(* IEC 61131-3 sources: MyTestRepos/BATTERY/PRG, 14 files *)

(* ---- PRG_AI.st ---- *)
PROGRAM PRG_AI
VAR
	F_Trig : ARRAY[1..cnst_num_ai] OF F_TRIG;
	i : INT;	(*Loop variable*)
	ManualFixChannels : BOOL; (*Will reset channels if faulty, i.e. card number is zero*)
	Reset: BOOL;
	Firstrun: BOOL;

	ai_CabinetTemperature_daemon: fb_AiProcess;
	ai_BatteryRoomTemperature_daemon: fb_AiProcess;
	ai_FilterTemperature_daemon: fb_AiProcess;

	ai_CabinetTemperature: str_AiProcess;
	ai_BatteryRoomTemperature: str_AiProcess;
	ai_FilterTemperature: str_AiProcess;

END_VAR

VAR RETAIN
	ai_CabinetTemperature_setup: str_AiSetup;
	ai_BatteryRoomTemperature_setup: str_AiSetup;
	ai_FilterTemperature_setup: str_AiSetup;
END_VAR

Reset := PRG_Functions.Reset;

(*Setup the HMI variables so that they are equal to actual used variables*)
IF (NOT Firstrun) THEN
	hmi_AiSetup[1] := ai_CabinetTemperature_setup;
	hmi_AiSetup[2] := ai_BatteryRoomTemperature_setup;
	hmi_AiSetup[3] := ai_FilterTemperature_setup;
	Firstrun := TRUE;
END_IF

(*Analog Input Signals*)
	ai_CabinetTemperature_daemon (setup:=ai_CabinetTemperature_setup,reset:=Reset,outPV=>ai_CabinetTemperature);
	ai_BatteryRoomTemperature_daemon (setup:=ai_BatteryRoomTemperature_setup,reset:=Reset,outPV=>ai_BatteryRoomTemperature);
	ai_FilterTemperature_daemon (setup:=ai_FilterTemperature_setup,reset:=Reset,outPV=>ai_FilterTemperature);

(*HMI Assign*)
	hmi_AiPV[1]:=ai_CabinetTemperature_daemon.outPV;
	hmi_AiPV[2]:=ai_BatteryRoomTemperature_daemon.outPV;
	hmi_AiPV[3]:=ai_FilterTemperature_daemon.outPV;

IF (ManualFixChannels) THEN  (*If manually forced: re-configure the channels*)
	FOR i:=0 TO cnst_num_ai BY 1 DO				(*Check if channel info is empty and restore if so.*)
		IF (PRG_HMI.setup_AioCard1_Number <> 0) THEN
			hmi_RestoreDefault_ai[i] := TRUE;
		END_IF
	END_FOR;
	ManualFixChannels := FALSE;
END_IF

END_PROGRAM

ACTIONS

ACTION Settings
(*
THIS SECTION CONTAINS HARD-CODED CHANNEL SETTINGS FOR EACH OF THE ANALOG INPUTS.

The settings are stored in retain memory, but whenever permanent changes are made, they should be hard coded into the appropriate channel below.
Each channel has settings for:

- Channel name (used for presentation in HMI)
- Channel- and card number (used to retrieve channel value via MIO lib)
- Channel type (4-20mA, PT100 etc)
- Channel forcing (force value and a bool flag to enable/disable forcing)
- Channel error flags, along with enable/disable flag + time delays
- Channel level flags, along with enable/disable flag + time delays

All setup values in retain memory can be forced to default (hard coded) values by setting RestoreAllToDefault,
or individually by setting hmi_RestoreDefault_ai[]. The latter is primary used from HMI.
*)
(***************ai_CabinetTemperature***************)
IF (RestoreAllToDefault OR ai_CabinetTemperature_setup.RestoreDefault  OR hmi_RestoreDefault_ai[1]) THEN
	ai_CabinetTemperature_setup.Name:='ai_CabinetTemperature';
	ai_CabinetTemperature_setup.CardNb:=PRG_HMI.setup_AioCard1_Number;
	ai_CabinetTemperature_setup.ChannelMode:=16#D3;
	ai_CabinetTemperature_setup.ChannelNb:=1;
 	ai_CabinetTemperature_setup.Enable.Forcing:=0;
 	ai_CabinetTemperature_setup.Enable.LLL:=0;
 	ai_CabinetTemperature_setup.Enable.LL:=0;
 	ai_CabinetTemperature_setup.Enable.L:=0;
 	ai_CabinetTemperature_setup.Enable.H:=0;
 	ai_CabinetTemperature_setup.Enable.HH:=0;
 	ai_CabinetTemperature_setup.Enable.HHH:=0;
 	ai_CabinetTemperature_setup.Enable.WireBreak:=1;
 	ai_CabinetTemperature_setup.Enable.Freeze:=1;
 	ai_CabinetTemperature_setup.Enable.High:=1;
 	ai_CabinetTemperature_setup.Enable.OOR:=1;
 	ai_CabinetTemperature_setup.Delay.LLL:=T#1s;
 	ai_CabinetTemperature_setup.Delay.LL:=T#1s;
 	ai_CabinetTemperature_setup.Delay.L:=T#1s;
 	ai_CabinetTemperature_setup.Delay.H:=T#1s;
 	ai_CabinetTemperature_setup.Delay.HH:=T#1s;
 	ai_CabinetTemperature_setup.Delay.HHH:=T#1s;
 	ai_CabinetTemperature_setup.Delay.WireBreak:=T#1s;
 	ai_CabinetTemperature_setup.Delay.High:=T#1s;
 	ai_CabinetTemperature_setup.Delay.OOR:=T#1s;
 	ai_CabinetTemperature_setup.Levels.LLL:=0;
 	ai_CabinetTemperature_setup.Levels.LL:=0;
 	ai_CabinetTemperature_setup.Levels.L:=0;
 	ai_CabinetTemperature_setup.Levels.H:=0;
 	ai_CabinetTemperature_setup.Levels.HH:=0;
 	ai_CabinetTemperature_setup.Levels.HHH:=0;
 	ai_CabinetTemperature_setup.Levels.Scale4mA:=0;
 	ai_CabinetTemperature_setup.Levels.Scale20mA:=100;
 	ai_CabinetTemperature_setup.Levels.ForceValue:=0;
END_IF
IF (hmi_RestoreDefault_ai[1] OR RestoreAllToDefault OR ai_CabinetTemperature_setup.RestoreDefault) THEN (*Copy values into HMI variable and reset*)
	hmi_AiSetup[1]:=ai_CabinetTemperature_setup; (*Copy setup values from retain into hmi variable*)
	hmi_RestoreDefault_ai[1]:=FALSE; (*Make sure that the restore variable is turned off after one restore command*)
	ai_CabinetTemperature_setup.RestoreDefault:=FALSE; (*Make sure that the restore variable is turned off after one restore command*)
END_IF
IF (hmi_AiWriteSetup[1]) THEN
	ai_CabinetTemperature_setup:=hmi_AiSetup[1]; (*Paste hmi changes back into setup variable*)
	hmi_AiWriteSetup[1]:=FALSE; (*Make sure that the write variable is turned off after one write command*)
END_IF
F_Trig[1](CLK:=hmi_AiPV[1].IsForced); (*Reset HMI forcing dialog when timer runs out*)
IF (F_Trig[1].Q) THEN hmi_AiSetup[1].Enable.Forcing:=FALSE;ai_CabinetTemperature_setup.Enable.Forcing:=FALSE; END_IF
(**************************************************)

(***************ai_BatteryRoomTemperature***************)
IF (RestoreAllToDefault OR ai_BatteryRoomTemperature_setup.RestoreDefault  OR hmi_RestoreDefault_ai[2]) THEN
	ai_BatteryRoomTemperature_setup.Name:='ai_BatteryRoomTemperature';
	ai_BatteryRoomTemperature_setup.CardNb:=PRG_HMI.setup_AioCard1_Number;
	ai_BatteryRoomTemperature_setup.ChannelMode:=16#D3;
	ai_BatteryRoomTemperature_setup.ChannelNb:=2;
 	ai_BatteryRoomTemperature_setup.Enable.Forcing:=0;
 	ai_BatteryRoomTemperature_setup.Enable.LLL:=0;
 	ai_BatteryRoomTemperature_setup.Enable.LL:=0;
 	ai_BatteryRoomTemperature_setup.Enable.L:=0;
 	ai_BatteryRoomTemperature_setup.Enable.H:=0;
 	ai_BatteryRoomTemperature_setup.Enable.HH:=0;
 	ai_BatteryRoomTemperature_setup.Enable.HHH:=0;
 	ai_BatteryRoomTemperature_setup.Enable.WireBreak:=1;
 	ai_BatteryRoomTemperature_setup.Enable.Freeze:=1;
 	ai_BatteryRoomTemperature_setup.Enable.High:=1;
 	ai_BatteryRoomTemperature_setup.Enable.OOR:=1;
 	ai_BatteryRoomTemperature_setup.Delay.LLL:=T#1s;
 	ai_BatteryRoomTemperature_setup.Delay.LL:=T#1s;
 	ai_BatteryRoomTemperature_setup.Delay.L:=T#1s;
 	ai_BatteryRoomTemperature_setup.Delay.H:=T#1s;
 	ai_BatteryRoomTemperature_setup.Delay.HH:=T#1s;
 	ai_BatteryRoomTemperature_setup.Delay.HHH:=T#1s;
 	ai_BatteryRoomTemperature_setup.Delay.WireBreak:=T#1s;
 	ai_BatteryRoomTemperature_setup.Delay.High:=T#1s;
 	ai_BatteryRoomTemperature_setup.Delay.OOR:=T#1s;
 	ai_BatteryRoomTemperature_setup.Levels.LLL:=0;
 	ai_BatteryRoomTemperature_setup.Levels.LL:=0;
 	ai_BatteryRoomTemperature_setup.Levels.L:=0;
 	ai_BatteryRoomTemperature_setup.Levels.H:=0;
 	ai_BatteryRoomTemperature_setup.Levels.HH:=0;
 	ai_BatteryRoomTemperature_setup.Levels.HHH:=0;
 	ai_BatteryRoomTemperature_setup.Levels.Scale4mA:=-20;
 	ai_BatteryRoomTemperature_setup.Levels.Scale20mA:=80;
 	ai_BatteryRoomTemperature_setup.Levels.ForceValue:=0;
END_IF
IF (hmi_RestoreDefault_ai[2] OR RestoreAllToDefault OR ai_BatteryRoomTemperature_setup.RestoreDefault) THEN (*Copy values into HMI variable and reset*)
	hmi_AiSetup[2]:=ai_BatteryRoomTemperature_setup; (*Copy setup values from retain into hmi variable*)
	hmi_RestoreDefault_ai[2]:=FALSE; (*Make sure that the restore variable is turned off after one restore command*)
	ai_BatteryRoomTemperature_setup.RestoreDefault:=FALSE; (*Make sure that the restore variable is turned off after one restore command*)
END_IF
IF (hmi_AiWriteSetup[2]) THEN
	ai_BatteryRoomTemperature_setup:=hmi_AiSetup[2]; (*Paste hmi changes back into setup variable*)
	hmi_AiWriteSetup[2]:=FALSE; (*Make sure that the write variable is turned off after one write command*)
END_IF
F_Trig[2](CLK:=hmi_AiPV[2].IsForced); (*Reset HMI forcing dialog when timer runs out*)
IF (F_Trig[2].Q) THEN hmi_AiSetup[2].Enable.Forcing:=FALSE;ai_BatteryRoomTemperature_setup.Enable.Forcing:=FALSE; END_IF
(**************************************************)

(***************ai_FilterTemperature***************)
IF (RestoreAllToDefault OR ai_FilterTemperature_setup.RestoreDefault  OR hmi_RestoreDefault_ai[3]) THEN
	ai_FilterTemperature_setup.Name:='ai_FilterTemperature';
	ai_FilterTemperature_setup.CardNb:=PRG_HMI.setup_AioCard1_Number;
	ai_FilterTemperature_setup.ChannelMode:=16#D1;
	ai_FilterTemperature_setup.ChannelNb:=4;
 	ai_FilterTemperature_setup.Enable.Forcing:=0;
 	ai_FilterTemperature_setup.Enable.LLL:=0;
 	ai_FilterTemperature_setup.Enable.LL:=0;
 	ai_FilterTemperature_setup.Enable.L:=0;
 	ai_FilterTemperature_setup.Enable.H:=0;
 	ai_FilterTemperature_setup.Enable.HH:=0;
 	ai_FilterTemperature_setup.Enable.HHH:=0;
 	ai_FilterTemperature_setup.Enable.WireBreak:=1;
 	ai_FilterTemperature_setup.Enable.Freeze:=1;
 	ai_FilterTemperature_setup.Enable.High:=1;
 	ai_FilterTemperature_setup.Enable.OOR:=1;
 	ai_FilterTemperature_setup.Delay.LLL:=T#1s;
 	ai_FilterTemperature_setup.Delay.LL:=T#1s;
 	ai_FilterTemperature_setup.Delay.L:=T#1s;
 	ai_FilterTemperature_setup.Delay.H:=T#1s;
 	ai_FilterTemperature_setup.Delay.HH:=T#1s;
 	ai_FilterTemperature_setup.Delay.HHH:=T#1s;
 	ai_FilterTemperature_setup.Delay.WireBreak:=T#1s;
 	ai_FilterTemperature_setup.Delay.High:=T#1s;
 	ai_FilterTemperature_setup.Delay.OOR:=T#1s;
 	ai_FilterTemperature_setup.Levels.LLL:=0;
 	ai_FilterTemperature_setup.Levels.LL:=0;
 	ai_FilterTemperature_setup.Levels.L:=0;
 	ai_FilterTemperature_setup.Levels.H:=0;
 	ai_FilterTemperature_setup.Levels.HH:=0;
 	ai_FilterTemperature_setup.Levels.HHH:=0;
 	ai_FilterTemperature_setup.Levels.Scale4mA:=0;
 	ai_FilterTemperature_setup.Levels.Scale20mA:=100;
 	ai_FilterTemperature_setup.Levels.ForceValue:=0;
END_IF
IF (hmi_RestoreDefault_ai[3] OR RestoreAllToDefault OR ai_FilterTemperature_setup.RestoreDefault) THEN (*Copy values into HMI variable and reset*)
	hmi_AiSetup[3]:=ai_FilterTemperature_setup; (*Copy setup values from retain into hmi variable*)
	hmi_RestoreDefault_ai[3]:=FALSE; (*Make sure that the restore variable is turned off after one restore command*)
	ai_FilterTemperature_setup.RestoreDefault:=FALSE; (*Make sure that the restore variable is turned off after one restore command*)
END_IF
IF (hmi_AiWriteSetup[3]) THEN
	ai_FilterTemperature_setup:=hmi_AiSetup[3]; (*Paste hmi changes back into setup variable*)
	hmi_AiWriteSetup[3]:=FALSE; (*Make sure that the write variable is turned off after one write command*)
END_IF
F_Trig[3](CLK:=hmi_AiPV[3].IsForced); (*Reset HMI forcing dialog when timer runs out*)
IF (F_Trig[3].Q) THEN hmi_AiSetup[3].Enable.Forcing:=FALSE;ai_FilterTemperature_setup.Enable.Forcing:=FALSE; END_IF
(**************************************************)

END_ACTION

END_ACTIONS

(* ---- PRG_Alarms.st ---- *)
PROGRAM PRG_Alarms
VAR
	pack: 					INT := 0;
	BMS_Alarm_Word: 		INT := 8; (*Must be first available word number after the ordinary alarms*)

	(*Two dimensional array for Set/Reset blocks. First index refers to word number (e.g. Alarmword[1]), second index refers to bit number*)
	AlarmSR: 				ARRAY[1..32,0..15] OF SR;
	Repeat_Alarm: 			fb_RepeatAlarm;
	Repeat_AlarmAppWarning:	fb_RepeatAlarm;
	E0AlarmWord:			fb_BitToWord;

	Reset : 				BOOL;
	CommonWarning: 			BOOL;
	CommonPLCWarning:		BOOL;
	CommonAppWarning:		BOOL;
	CommonIoWarning:		BOOL;
	CommonLevelWarning:		BOOL;
	CommonSignalWarning:	BOOL;
	CommonE0Warning:		BOOL;
END_VAR

Reset := PRG_Functions.Reset;

(*Gorup alarms with blinking on new alarms within their group*)
CommonWarning :=  		Repeat_Alarm.Alarm_common;
CommonPLCWarning := 	Repeat_Alarm.Alarm_Repeat1;
CommonSignalWarning:= 	Repeat_Alarm.Alarm_Repeat2;
CommonIoWarning	 := 	Repeat_Alarm.Alarm_Repeat3;
CommonLevelWarning := 	Repeat_Alarm.Alarm_Repeat4;
CommonAppWarning := 	Repeat_AlarmAppWarning.Alarm_common;
CommonE0Warning := 		Repeat_Alarm.Alarm_Repeat20;

(*Single alarms used for E0 *)
E0AlarmWord(
	EN := TRUE,
	Bit0 := PRG_DI.di_WaterLeakageDetected.PV,
	Bit1 := PRG_BatteryProtection.batteryPreWarning,
	Bit2 := PRG_BatteryProtection.Warning_CellTemp_L,
	Bit3 := PRG_BatteryProtection.Warning_CellVolt_L_Offline,
	Bit4 := PRG_BatteryProtection.Warning_CellVolt_LL_Offline,
	Bit5 := PRG_BatteryProtection.Warning_SoC_L_Offline,
	Bit6 := FALSE,
	Bit7 := FALSE,
	Bit8 := FALSE,
	Bit9 := FALSE,
	Bit10 := FALSE,
	Bit11 := FALSE,
	Bit12 := FALSE,
	Bit13 := FALSE,
	Bit14 := FALSE,
	Bit15 := FALSE,
	OUT =>
);

(*General PLC warnings*)
AlarmSR[1,0] (SET1:=(PRG_HW.HwAlarmCPU.AlarmCpuLoad) ,  Q1=>AlarmWord[1].0, RESET:=PRG_Functions.Reset);(*High Load on CPU*)
AlarmSR[1,1] (SET1:=(PRG_HW.HwAlarmCPU.AlarmCpuTemp) ,  Q1=>AlarmWord[1].1, RESET:=PRG_Functions.Reset);(*High Temperature on CPU*)
AlarmSR[1,2] (SET1:=(PRG_HW.HwAlarmCPU.AlarmFreeMem) ,  Q1=>AlarmWord[1].2, RESET:=PRG_Functions.Reset);(*Low Free Memory on PLC CPU*)
AlarmSR[1,3] (SET1:=(PRG_HW.Em0In.Alarm) ,  Q1=>AlarmWord[1].3, RESET:=PRG_Functions.Reset);(*High Load on EM213 Network Card*)
AlarmSR[1,4] (SET1:=(PRG_HW.Eth0In.Alarm) ,  Q1=>AlarmWord[1].4, RESET:=PRG_Functions.Reset);(*High Load on Ethernet Port ETH1*)
AlarmSR[1,5] (SET1:=(PRG_HW.Eth1In.Alarm) ,  Q1=>AlarmWord[1].5, RESET:=PRG_Functions.Reset);(*High Load on Ethernet Port ETH2*)

(*Signal warnings, OOR and wirebreak etc*)
AlarmSR[2,0] (SET1:=(PRG_AI.ai_BatteryRoomTemperature.Alarm.common) ,  Q1=>AlarmWord[2].0, RESET:=PRG_Functions.Reset);(*Battery Room Temperature - 4mA loop fail*)
AlarmSR[2,1] (SET1:=(PRG_AI.ai_CabinetTemperature.Alarm.common) ,  Q1=>AlarmWord[2].1, RESET:=PRG_Functions.Reset);(*Cabinet Temperature - Loop Failure*)
AlarmSR[2,2] (SET1:=(PRG_AI.ai_FilterTemperature.Alarm.common) ,  Q1=>AlarmWord[2].2, RESET:=PRG_Functions.Reset);(*LC Filter Temperature - Loop Failure*)
AlarmSR[2,3] (SET1:=(PRG_AO.ao_BatteryCurrentInstr.Alarm.common) ,  Q1=>AlarmWord[2].3, RESET:=PRG_Functions.Reset);(*Current Instrument 4-20mA Loop Failure*)
AlarmSR[2,4] (SET1:=(PRG_AO.ao_BatteryPowerInstr.Alarm.common) ,  Q1=>AlarmWord[2].4, RESET:=PRG_Functions.Reset);(*Power Instrument 4-20mA Loop Failure*)
AlarmSR[2,5] (SET1:=(PRG_AO.ao_BatteryVoltageInstr.Alarm.common) ,  Q1=>AlarmWord[2].5, RESET:=PRG_Functions.Reset);(*Voltage Instrument 4-20mA Loop Failure*)
AlarmSR[2,6] (SET1:=(PRG_AO.ao_BatterySocInstr.Alarm.common) ,  Q1=>AlarmWord[2].6, RESET:=PRG_Functions.Reset);(*SoC Instrument 4-20mA Loop Failure*)
AlarmSR[2,7] (SET1:=(PRG_AO.ao_BatteryChrgDischrgInstr.Alarm.common) ,  Q1=>AlarmWord[2].7, RESET:=PRG_Functions.Reset);(*Charge/Discharge Instrument 4-20mA Loop Failure*)

(*IO warnings, alarm contacts, module error etc*)
AlarmSR[3,0] (SET1:=(PRG_HW.AioCardError1) ,  Q1=>AlarmWord[3].0, RESET:=PRG_Functions.Reset);(*Common Alarm from PLC I/O Analog IO Card*)
AlarmSR[3,1] (SET1:=(PRG_HW.DioCardError1) ,  Q1=>AlarmWord[3].1, RESET:=PRG_Functions.Reset);(*Common Alarm from PLC I/O Digital IO Card*)
AlarmSR[3,2] (SET1:=(PRG_Functions.Breaker.Alarm_delayed) ,  Q1=>AlarmWord[3].2, RESET:=PRG_Functions.Reset);(*Voting Alarm DC Breaker Position*)
AlarmSR[3,3] (SET1:=(PRG_DI.di_EmergencyStopLoopFault.PV) ,  Q1=>AlarmWord[3].3, RESET:=PRG_Functions.Reset);(*Emergency Stop Loop Alarm*)
AlarmSR[3,4] (SET1:=(PRG_Operation.ControlPlace.alarmDeviation) ,  Q1=>AlarmWord[3].4, RESET:=PRG_Functions.Reset);(*Voting Alarm Local/Remote Switch*)
AlarmSR[3,5] (SET1:=(NOT PRG_DI.di_EthernetSwitchAlarm.PV AND PRG_HMI.enEthernetSwitchAlarm) ,  Q1=>AlarmWord[3].5, RESET:=PRG_Functions.Reset);(*External Ethernet Switch Alarm*)

(*Level warning, high or low etc*)
AlarmSR[4,0] (SET1:=(PRG_AI.ai_BatteryRoomTemperature.Alarm.HH) ,  Q1=>AlarmWord[4].0, RESET:=PRG_Functions.Reset);(*Battery Room High Temperature*)
AlarmSR[4,1] (SET1:=(PRG_AI.ai_BatteryRoomTemperature.Alarm.LL) ,  Q1=>AlarmWord[4].1, RESET:=PRG_Functions.Reset);(*Battery Room Low Temperature*)
AlarmSR[4,2] (SET1:=(PRG_AI.ai_BatteryRoomTemperature.Alarm.HHH) ,  Q1=>AlarmWord[4].2, RESET:=PRG_Functions.Reset);(*Battery Room HighHigh Temperature*)
AlarmSR[4,3] (SET1:=(PRG_AI.ai_BatteryRoomTemperature.Alarm.LLL) ,  Q1=>AlarmWord[4].3, RESET:=PRG_Functions.Reset);(*Battery Room LowLow Temperature*)
AlarmSR[4,4] (SET1:=(PRG_AI.ai_CabinetTemperature.Alarm.HH) ,  Q1=>AlarmWord[4].4, RESET:=PRG_Functions.Reset);(*Cabinet High Temperature*)
AlarmSR[4,5] (SET1:=(PRG_AI.ai_CabinetTemperature.Alarm.LL) ,  Q1=>AlarmWord[4].5, RESET:=PRG_Functions.Reset);(*Cabinet Low Temperature*)
AlarmSR[4,6] (SET1:=(PRG_AI.ai_FilterTemperature.Alarm.HH) ,  Q1=>AlarmWord[4].6, RESET:=PRG_Functions.Reset);(*LC Filter High Temperature*)
AlarmSR[4,7] (SET1:=(PRG_AI.ai_FilterTemperature.Alarm.LL) ,  Q1=>AlarmWord[4].7, RESET:=PRG_Functions.Reset);(*LC Filter Low Temperature*)
AlarmSR[4,8] (SET1:=(PRG_Drive.UnitOverTempAlarm) ,  Q1=>AlarmWord[4].8, RESET:=PRG_Functions.Reset);(*Vacon Unit High Temperature*)

(*Application specific warnings*)
AlarmSR[5,0] (SET1:=(PRG_Drive.Status.Warning) ,  Q1=>AlarmWord[5].0, RESET:=PRG_Functions.Reset);(*Common Alarm from DC/DC Converter*)
AlarmSR[5,1] (SET1:=(PRG_BatteryProtection.batteryCommonWarning) ,  Q1=>AlarmWord[5].1, RESET:=PRG_Functions.Reset);(*Common Alarm from Battery Management System*)
AlarmSR[5,2] (SET1:=(PRG_StateMain.StartingTimeout) ,  Q1=>AlarmWord[5].2, RESET:=PRG_Functions.Reset);(*Start Sequence Timeout*)
AlarmSR[5,3] (SET1:=(PRG_StateMain.StoppingTimeout) ,  Q1=>AlarmWord[5].3, RESET:=PRG_Functions.Reset);(*Stop Sequence Timeout - Failsafe Trip*)
AlarmSR[5,4] (SET1:=(PRG_DI.di_WaterLeakageDetected.PV) ,  Q1=>AlarmWord[5].4, RESET:=PRG_Functions.Reset);(*Water Leakage in DC/DC Section*)
AlarmSR[5,5] (SET1:=(PRG_Battery.StopChargeTOF.Q) ,  Q1=>AlarmWord[5].5, RESET:=PRG_Functions.Reset);(*Battery Charge Limit in Effect*)
AlarmSR[5,6] (SET1:=(PRG_Battery.StopDischargeTOF.Q) ,  Q1=>AlarmWord[5].6, RESET:=PRG_Functions.Reset);(*Battery Discharge Limit in Effect*)
AlarmSR[5,7] (SET1:=(NOT PRG_Functions.Breaker.DI_Verif_delay OR NOT PRG_DI.di_DcBreakerEarlyBreak.PV) ,  Q1=>AlarmWord[5].7, RESET:=PRG_Functions.Reset);(*DC Breaker Open - Start Inhibited*)
AlarmSR[5,8] (SET1:=(PRG_Operation.ControlPlace.ctrlLocation = e_Local) ,  Q1=>AlarmWord[5].8, RESET:=PRG_Functions.Reset);(*In Local Control*)
AlarmSR[5,9] (SET1:=(PRG_IAS.IasCommunication.Alarm) ,  Q1=>AlarmWord[5].9, RESET:=PRG_Functions.Reset);(*IAS Communication Alarm*)
AlarmSR[5,10] (SET1:=(PRG_BatteryComm.NoPrechargePackComm) ,  Q1=>AlarmWord[5].10, RESET:=PRG_Functions.Reset);(*Comm. Failure Battery Precharge System*)
AlarmSR[5,11] (SET1:=((PRG_StateMain.RunningTON.Q) AND NOT PRG_Battery.BatteryAllConnected) ,  Q1=>AlarmWord[5].11, RESET:=PRG_Functions.Reset);(*All Batteries are not Connected*)
AlarmSR[5,12] (SET1:=(PRG_StateMain.BatteryConnectionTimeout) ,  Q1=>AlarmWord[5].12, RESET:=PRG_Functions.Reset);(*Battery Connection Timeout during Starting*)
AlarmSR[5,13] (SET1:=(PRG_StateMain.BatteryDisconnectionTimeout) ,  Q1=>AlarmWord[5].13, RESET:=PRG_Functions.Reset);(*Battery Disconnection Timeout during Stopping*)

(*Battery Specific PLC Alarms*)
AlarmSR[6,0] (SET1:=(PRG_BatteryProtection.batteryPreWarning) ,  Q1=>AlarmWord[6].0, RESET:=PRG_Functions.Reset);(*Prewarning from Battery Management System*)
AlarmSR[6,1] (SET1:=(PRG_BatteryProtection.Warning_SoC_L) ,  Q1=>AlarmWord[6].1, RESET:=PRG_Functions.Reset);(*State of Charge Low Alarm - Start Charging*)
AlarmSR[6,2] (SET1:=(PRG_BatteryProtection.Warning_SoC_H) ,  Q1=>AlarmWord[6].2, RESET:=PRG_Functions.Reset);(*State of Charge High Alarm*)
AlarmSR[6,3] (SET1:=(PRG_BatteryProtection.Warning_Volt_H) ,  Q1=>AlarmWord[6].3, RESET:=PRG_Functions.Reset);(*High Battery Voltage Alarm*)
AlarmSR[6,4] (SET1:=(PRG_BatteryProtection.Warning_Volt_L) ,  Q1=>AlarmWord[6].4, RESET:=PRG_Functions.Reset);(*Low Battery Voltage Alarm*)
AlarmSR[6,5] (SET1:=(PRG_BatteryProtection.Warning_CellVolt_L) ,  Q1=>AlarmWord[6].5, RESET:=PRG_Functions.Reset);(*Low Cell Voltage Alarm*)
AlarmSR[6,6] (SET1:=(PRG_BatteryProtection.Warning_CellVolt_H) ,  Q1=>AlarmWord[6].6, RESET:=PRG_Functions.Reset);(*High Cell Voltage Alarm*)
AlarmSR[6,7] (SET1:=(PRG_BatteryProtection.Warning_CellTemp_L) ,  Q1=>AlarmWord[6].7, RESET:=PRG_Functions.Reset);(*Low Cell Temperature Alarm*)
AlarmSR[6,8] (SET1:=(PRG_BatteryProtection.Warning_CellTemp_H) ,  Q1=>AlarmWord[6].8, RESET:=PRG_Functions.Reset);(*High Cell Temperature Alarm*)
AlarmSR[6,9] (SET1:=(PRG_BatteryProtection.Warning_SoC_L_Offline) ,  Q1=>AlarmWord[6].9, RESET:=PRG_Functions.Reset);(*Offline Low SoC: Connect and Charge Now*)
AlarmSR[6,10] (SET1:=(PRG_BatteryProtection.Warning_CellVolt_L_Offline) ,  Q1=>AlarmWord[6].10, RESET:=PRG_Functions.Reset);(*Offline Low Cell Voltage: Connect and Charge Now*)
AlarmSR[6,11] (SET1:=(PRG_BatteryProtection.Warning_CellVolt_LL_Offline) ,  Q1=>AlarmWord[6].11, RESET:=PRG_Functions.Reset);(*Offline Low Cell Voltage: Critical Level - Charge Now*)
AlarmSR[6,12] (SET1:=(PRG_HMI.SoHVerifModeActive) ,  Q1=>AlarmWord[6].12, RESET:=PRG_Functions.Reset);(*SoH Verification Mode Active: SoC Limits Extended*)

(*Auto generated alarms from Corvus BMS*)

BMS_Alarm_Word:= 8; (*Next available alarmword*)
FOR pack := 1 TO DINT_TO_INT(PRG_HMI.setup_Battery_total_nr_of_packs) BY 1 DO
	AlarmSR[BMS_Alarm_Word,0] (SET1:=(PRG_BatteryComm.CorvusRead[pack].FW.Input_PowerLoss_Warning) ,  Q1=>AlarmWord[BMS_Alarm_Word].0, RESET:=Reset);(*BMS Pack  Input Power Loss Warning*)
	AlarmSR[BMS_Alarm_Word,1] (SET1:=(PRG_BatteryComm.CorvusRead[pack].FW.Module_Communication_Warning) ,  Q1=>AlarmWord[BMS_Alarm_Word].1, RESET:=Reset);(*BMS Pack  Module Communication Warning*)
	AlarmSR[BMS_Alarm_Word,2] (SET1:=(PRG_BatteryComm.CorvusRead[pack].FW.OverCurrent_Warning) ,  Q1=>AlarmWord[BMS_Alarm_Word].2, RESET:=Reset);(*BMS Pack  Over Current Warning*)
	AlarmSR[BMS_Alarm_Word,3] (SET1:=(PRG_BatteryComm.CorvusRead[pack].FW.PDM_overTemperature_Warning) ,  Q1=>AlarmWord[BMS_Alarm_Word].3, RESET:=Reset);(*BMS Pack  PDM Over Temperature Warning*)
	AlarmSR[BMS_Alarm_Word,4] (SET1:=(PRG_BatteryComm.CorvusRead[pack].FW.SE_overTemperature_Warning) ,  Q1=>AlarmWord[BMS_Alarm_Word].4, RESET:=Reset);(*BMS Pack  Cell Over Temperature Warning*)
	AlarmSR[BMS_Alarm_Word,5] (SET1:=(PRG_BatteryComm.CorvusRead[pack].FW.SE_overVoltage_Warning) ,  Q1=>AlarmWord[BMS_Alarm_Word].5, RESET:=Reset);(*BMS Pack  Cell Over Voltage Warning*)
	AlarmSR[BMS_Alarm_Word,6] (SET1:=(PRG_BatteryComm.CorvusRead[pack].FW.SE_underVoltage_Warning) ,  Q1=>AlarmWord[BMS_Alarm_Word].6, RESET:=Reset);(*BMS Pack  Cell Under Voltage Warning*)
	AlarmSR[BMS_Alarm_Word,7] (SET1:=(PRG_BatteryComm.CorvusRead[pack].ModbusFault AND NOT PRG_BatteryComm.CorvusBMS_Total_Comm_Fault) ,  Q1=>AlarmWord[BMS_Alarm_Word].7, RESET:=Reset);(*BMS Pack Communication Alarm*)
	BMS_Alarm_Word :=  BMS_Alarm_Word+1;
END_FOR

(*Blinks the alarm output*)

Repeat_AlarmAppWarning(
	AlarmWord5:= INT_TO_WORD(AlarmWord[5]),
	AlarmWord6:= INT_TO_WORD(AlarmWord[6]),
);

Repeat_Alarm(
	AlarmWord1:= INT_TO_WORD(AlarmWord[1]),
	AlarmWord2:= INT_TO_WORD(AlarmWord[2]),
	AlarmWord3:= INT_TO_WORD(AlarmWord[3]),
	AlarmWord4:= INT_TO_WORD(AlarmWord[4]),
	AlarmWord5:= INT_TO_WORD(AlarmWord[5]),
	AlarmWord6:= INT_TO_WORD(AlarmWord[6]),
	AlarmWord7:= INT_TO_WORD(AlarmWord[7]),
	AlarmWord8:= INT_TO_WORD(AlarmWord[8]),
	AlarmWord9:= INT_TO_WORD(AlarmWord[9]),
	AlarmWord10:= INT_TO_WORD(AlarmWord[10]),
	AlarmWord11:= INT_TO_WORD(AlarmWord[11]),
	AlarmWord12:= INT_TO_WORD(AlarmWord[12]),
	AlarmWord13:= INT_TO_WORD(AlarmWord[13]),
	AlarmWord14:= INT_TO_WORD(AlarmWord[14]),
	AlarmWord15:= INT_TO_WORD(AlarmWord[15]),
	AlarmWord16:= INT_TO_WORD(AlarmWord[16]),
	AlarmWord17:= INT_TO_WORD(AlarmWord[17]),
	AlarmWord18:= INT_TO_WORD(AlarmWord[18]),
	AlarmWord19:= INT_TO_WORD(AlarmWord[19]),
	AlarmWord20:= DINT_TO_WORD(E0AlarmWord.OUT),
	Alarm_common => ,
	Alarm_count => ,
	Alarm_Repeat1 => ,
	Alarm_Repeat2 => ,
	Alarm_Repeat3 => ,
	Alarm_Repeat4 => ,
	Alarm_Repeat5 => ,
	Alarm_Repeat6 => ,
	Alarm_Repeat7 => ,
	Alarm_Repeat8 => ,
	Alarm_Repeat9 => ,
	Alarm_Repeat10 => ,
	Alarm_Repeat11 => ,
	Alarm_Repeat12 => ,
	Alarm_Repeat13 => ,
	Alarm_Repeat14 => ,
	Alarm_Repeat15 => ,
	Alarm_Repeat16 => ,
	Alarm_Repeat17 => ,
	Alarm_Repeat18 => ,
	Alarm_Repeat19 => ,
	Alarm_Repeat20 =>
);

END_PROGRAM

ACTIONS
ACTION hmi_Alarms
hmi_AlarmWord[1].0 := AlarmSR[1,0].Q1;
hmi_AlarmWord[1].1 := AlarmSR[1,1].Q1;
hmi_AlarmWord[1].2 := AlarmSR[1,2].Q1;
hmi_AlarmWord[1].3 := AlarmSR[1,3].Q1;
hmi_AlarmWord[1].4 := AlarmSR[1,4].Q1;
hmi_AlarmWord[1].5 := AlarmSR[1,5].Q1;
hmi_AlarmWord[1].6 := AlarmSR[1,6].Q1;
hmi_AlarmWord[1].7 := AlarmSR[1,7].Q1;
hmi_AlarmWord[1].8 := AlarmSR[1,8].Q1;
hmi_AlarmWord[1].9 := AlarmSR[1,9].Q1;
hmi_AlarmWord[1].10 := AlarmSR[1,10].Q1;
hmi_AlarmWord[1].11 := AlarmSR[1,11].Q1;
hmi_AlarmWord[1].12 := AlarmSR[1,12].Q1;
hmi_AlarmWord[1].13 := AlarmSR[1,13].Q1;
hmi_AlarmWord[1].14 := AlarmSR[1,14].Q1;
hmi_AlarmWord[1].15 := AlarmSR[1,15].Q1;
hmi_AlarmWord[2].0 := AlarmSR[2,0].Q1;
hmi_AlarmWord[2].1 := AlarmSR[2,1].Q1;
hmi_AlarmWord[2].2 := AlarmSR[2,2].Q1;
hmi_AlarmWord[2].3 := AlarmSR[2,3].Q1;
hmi_AlarmWord[2].4 := AlarmSR[2,4].Q1;
hmi_AlarmWord[2].5 := AlarmSR[2,5].Q1;
hmi_AlarmWord[2].6 := AlarmSR[2,6].Q1;
hmi_AlarmWord[2].7 := AlarmSR[2,7].Q1;
hmi_AlarmWord[2].8 := AlarmSR[2,8].Q1;
hmi_AlarmWord[2].9 := AlarmSR[2,9].Q1;
hmi_AlarmWord[2].10 := AlarmSR[2,10].Q1;
hmi_AlarmWord[2].11 := AlarmSR[2,11].Q1;
hmi_AlarmWord[2].12 := AlarmSR[2,12].Q1;
hmi_AlarmWord[2].13 := AlarmSR[2,13].Q1;
hmi_AlarmWord[2].14 := AlarmSR[2,14].Q1;
hmi_AlarmWord[2].15 := AlarmSR[2,15].Q1;
hmi_AlarmWord[3].0 := AlarmSR[3,0].Q1;
hmi_AlarmWord[3].1 := AlarmSR[3,1].Q1;
hmi_AlarmWord[3].2 := AlarmSR[3,2].Q1;
hmi_AlarmWord[3].3 := AlarmSR[3,3].Q1;
hmi_AlarmWord[3].4 := AlarmSR[3,4].Q1;
hmi_AlarmWord[3].5 := AlarmSR[3,5].Q1;
hmi_AlarmWord[3].6 := AlarmSR[3,6].Q1;
hmi_AlarmWord[3].7 := AlarmSR[3,7].Q1;
hmi_AlarmWord[3].8 := AlarmSR[3,8].Q1;
hmi_AlarmWord[3].9 := AlarmSR[3,9].Q1;
hmi_AlarmWord[3].10 := AlarmSR[3,10].Q1;
hmi_AlarmWord[3].11 := AlarmSR[3,11].Q1;
hmi_AlarmWord[3].12 := AlarmSR[3,12].Q1;
hmi_AlarmWord[3].13 := AlarmSR[3,13].Q1;
hmi_AlarmWord[3].14 := AlarmSR[3,14].Q1;
hmi_AlarmWord[3].15 := AlarmSR[3,15].Q1;
hmi_AlarmWord[4].0 := AlarmSR[4,0].Q1;
hmi_AlarmWord[4].1 := AlarmSR[4,1].Q1;
hmi_AlarmWord[4].2 := AlarmSR[4,2].Q1;
hmi_AlarmWord[4].3 := AlarmSR[4,3].Q1;
hmi_AlarmWord[4].4 := AlarmSR[4,4].Q1;
hmi_AlarmWord[4].5 := AlarmSR[4,5].Q1;
hmi_AlarmWord[4].6 := AlarmSR[4,6].Q1;
hmi_AlarmWord[4].7 := AlarmSR[4,7].Q1;
hmi_AlarmWord[4].8 := AlarmSR[4,8].Q1;
hmi_AlarmWord[4].9 := AlarmSR[4,9].Q1;
hmi_AlarmWord[4].10 := AlarmSR[4,10].Q1;
hmi_AlarmWord[4].11 := AlarmSR[4,11].Q1;
hmi_AlarmWord[4].12 := AlarmSR[4,12].Q1;
hmi_AlarmWord[4].13 := AlarmSR[4,13].Q1;
hmi_AlarmWord[4].14 := AlarmSR[4,14].Q1;
hmi_AlarmWord[4].15 := AlarmSR[4,15].Q1;
hmi_AlarmWord[5].0 := AlarmSR[5,0].Q1;
hmi_AlarmWord[5].1 := AlarmSR[5,1].Q1;
hmi_AlarmWord[5].2 := AlarmSR[5,2].Q1;
hmi_AlarmWord[5].3 := AlarmSR[5,3].Q1;
hmi_AlarmWord[5].4 := AlarmSR[5,4].Q1;
hmi_AlarmWord[5].5 := AlarmSR[5,5].Q1;
hmi_AlarmWord[5].6 := AlarmSR[5,6].Q1;
hmi_AlarmWord[5].7 := AlarmSR[5,7].Q1;
hmi_AlarmWord[5].8 := AlarmSR[5,8].Q1;
hmi_AlarmWord[5].9 := AlarmSR[5,9].Q1;
hmi_AlarmWord[5].10 := AlarmSR[5,10].Q1;
hmi_AlarmWord[5].11 := AlarmSR[5,11].Q1;
hmi_AlarmWord[5].12 := AlarmSR[5,12].Q1;
hmi_AlarmWord[5].13 := AlarmSR[5,13].Q1;
hmi_AlarmWord[5].14 := AlarmSR[5,14].Q1;
hmi_AlarmWord[5].15 := AlarmSR[5,15].Q1;
hmi_AlarmWord[6].0 := AlarmSR[6,0].Q1;
hmi_AlarmWord[6].1 := AlarmSR[6,1].Q1;
hmi_AlarmWord[6].2 := AlarmSR[6,2].Q1;
hmi_AlarmWord[6].3 := AlarmSR[6,3].Q1;
hmi_AlarmWord[6].4 := AlarmSR[6,4].Q1;
hmi_AlarmWord[6].5 := AlarmSR[6,5].Q1;
hmi_AlarmWord[6].6 := AlarmSR[6,6].Q1;
hmi_AlarmWord[6].7 := AlarmSR[6,7].Q1;
hmi_AlarmWord[6].8 := AlarmSR[6,8].Q1;
hmi_AlarmWord[6].9 := AlarmSR[6,9].Q1;
hmi_AlarmWord[6].10 := AlarmSR[6,10].Q1;
hmi_AlarmWord[6].11 := AlarmSR[6,11].Q1;
hmi_AlarmWord[6].12 := AlarmSR[6,12].Q1;
hmi_AlarmWord[6].13 := AlarmSR[6,13].Q1;
hmi_AlarmWord[6].14 := AlarmSR[6,14].Q1;
hmi_AlarmWord[6].15 := AlarmSR[6,15].Q1;
hmi_AlarmWord[7].0 := AlarmSR[7,0].Q1;
hmi_AlarmWord[7].1 := AlarmSR[7,1].Q1;
hmi_AlarmWord[7].2 := AlarmSR[7,2].Q1;
hmi_AlarmWord[7].3 := AlarmSR[7,3].Q1;
hmi_AlarmWord[7].4 := AlarmSR[7,4].Q1;
hmi_AlarmWord[7].5 := AlarmSR[7,5].Q1;
hmi_AlarmWord[7].6 := AlarmSR[7,6].Q1;
hmi_AlarmWord[7].7 := AlarmSR[7,7].Q1;
hmi_AlarmWord[7].8 := AlarmSR[7,8].Q1;
hmi_AlarmWord[7].9 := AlarmSR[7,9].Q1;
hmi_AlarmWord[7].10 := AlarmSR[7,10].Q1;
hmi_AlarmWord[7].11 := AlarmSR[7,11].Q1;
hmi_AlarmWord[7].12 := AlarmSR[7,12].Q1;
hmi_AlarmWord[7].13 := AlarmSR[7,13].Q1;
hmi_AlarmWord[7].14 := AlarmSR[7,14].Q1;
hmi_AlarmWord[7].15 := AlarmSR[7,15].Q1;
hmi_AlarmWord[8].0 := AlarmSR[8,0].Q1;
hmi_AlarmWord[8].1 := AlarmSR[8,1].Q1;
hmi_AlarmWord[8].2 := AlarmSR[8,2].Q1;
hmi_AlarmWord[8].3 := AlarmSR[8,3].Q1;
hmi_AlarmWord[8].4 := AlarmSR[8,4].Q1;
hmi_AlarmWord[8].5 := AlarmSR[8,5].Q1;
hmi_AlarmWord[8].6 := AlarmSR[8,6].Q1;
hmi_AlarmWord[8].7 := AlarmSR[8,7].Q1;
hmi_AlarmWord[8].8 := AlarmSR[8,8].Q1;
hmi_AlarmWord[8].9 := AlarmSR[8,9].Q1;
hmi_AlarmWord[8].10 := AlarmSR[8,10].Q1;
hmi_AlarmWord[8].11 := AlarmSR[8,11].Q1;
hmi_AlarmWord[8].12 := AlarmSR[8,12].Q1;
hmi_AlarmWord[8].13 := AlarmSR[8,13].Q1;
hmi_AlarmWord[8].14 := AlarmSR[8,14].Q1;
hmi_AlarmWord[8].15 := AlarmSR[8,15].Q1;
hmi_AlarmWord[9].0 := AlarmSR[9,0].Q1;
hmi_AlarmWord[9].1 := AlarmSR[9,1].Q1;
hmi_AlarmWord[9].2 := AlarmSR[9,2].Q1;
hmi_AlarmWord[9].3 := AlarmSR[9,3].Q1;
hmi_AlarmWord[9].4 := AlarmSR[9,4].Q1;
hmi_AlarmWord[9].5 := AlarmSR[9,5].Q1;
hmi_AlarmWord[9].6 := AlarmSR[9,6].Q1;
hmi_AlarmWord[9].7 := AlarmSR[9,7].Q1;
hmi_AlarmWord[9].8 := AlarmSR[9,8].Q1;
hmi_AlarmWord[9].9 := AlarmSR[9,9].Q1;
hmi_AlarmWord[9].10 := AlarmSR[9,10].Q1;
hmi_AlarmWord[9].11 := AlarmSR[9,11].Q1;
hmi_AlarmWord[9].12 := AlarmSR[9,12].Q1;
hmi_AlarmWord[9].13 := AlarmSR[9,13].Q1;
hmi_AlarmWord[9].14 := AlarmSR[9,14].Q1;
hmi_AlarmWord[9].15 := AlarmSR[9,15].Q1;
hmi_AlarmWord[10].0 := AlarmSR[10,0].Q1;
hmi_AlarmWord[10].1 := AlarmSR[10,1].Q1;
hmi_AlarmWord[10].2 := AlarmSR[10,2].Q1;
hmi_AlarmWord[10].3 := AlarmSR[10,3].Q1;
hmi_AlarmWord[10].4 := AlarmSR[10,4].Q1;
hmi_AlarmWord[10].5 := AlarmSR[10,5].Q1;
hmi_AlarmWord[10].6 := AlarmSR[10,6].Q1;
hmi_AlarmWord[10].7 := AlarmSR[10,7].Q1;
hmi_AlarmWord[10].8 := AlarmSR[10,8].Q1;
hmi_AlarmWord[10].9 := AlarmSR[10,9].Q1;
hmi_AlarmWord[10].10 := AlarmSR[10,10].Q1;
hmi_AlarmWord[10].11 := AlarmSR[10,11].Q1;
hmi_AlarmWord[10].12 := AlarmSR[10,12].Q1;
hmi_AlarmWord[10].13 := AlarmSR[10,13].Q1;
hmi_AlarmWord[10].14 := AlarmSR[10,14].Q1;
hmi_AlarmWord[10].15 := AlarmSR[10,15].Q1;
hmi_AlarmWord[11].0 := AlarmSR[11,0].Q1;
hmi_AlarmWord[11].1 := AlarmSR[11,1].Q1;
hmi_AlarmWord[11].2 := AlarmSR[11,2].Q1;
hmi_AlarmWord[11].3 := AlarmSR[11,3].Q1;
hmi_AlarmWord[11].4 := AlarmSR[11,4].Q1;
hmi_AlarmWord[11].5 := AlarmSR[11,5].Q1;
hmi_AlarmWord[11].6 := AlarmSR[11,6].Q1;
hmi_AlarmWord[11].7 := AlarmSR[11,7].Q1;
hmi_AlarmWord[11].8 := AlarmSR[11,8].Q1;
hmi_AlarmWord[11].9 := AlarmSR[11,9].Q1;
hmi_AlarmWord[11].10 := AlarmSR[11,10].Q1;
hmi_AlarmWord[11].11 := AlarmSR[11,11].Q1;
hmi_AlarmWord[11].12 := AlarmSR[11,12].Q1;
hmi_AlarmWord[11].13 := AlarmSR[11,13].Q1;
hmi_AlarmWord[11].14 := AlarmSR[11,14].Q1;
hmi_AlarmWord[11].15 := AlarmSR[11,15].Q1;
hmi_AlarmWord[12].0 := AlarmSR[12,0].Q1;
hmi_AlarmWord[12].1 := AlarmSR[12,1].Q1;
hmi_AlarmWord[12].2 := AlarmSR[12,2].Q1;
hmi_AlarmWord[12].3 := AlarmSR[12,3].Q1;
hmi_AlarmWord[12].4 := AlarmSR[12,4].Q1;
hmi_AlarmWord[12].5 := AlarmSR[12,5].Q1;
hmi_AlarmWord[12].6 := AlarmSR[12,6].Q1;
hmi_AlarmWord[12].7 := AlarmSR[12,7].Q1;
hmi_AlarmWord[12].8 := AlarmSR[12,8].Q1;
hmi_AlarmWord[12].9 := AlarmSR[12,9].Q1;
hmi_AlarmWord[12].10 := AlarmSR[12,10].Q1;
hmi_AlarmWord[12].11 := AlarmSR[12,11].Q1;
hmi_AlarmWord[12].12 := AlarmSR[12,12].Q1;
hmi_AlarmWord[12].13 := AlarmSR[12,13].Q1;
hmi_AlarmWord[12].14 := AlarmSR[12,14].Q1;
hmi_AlarmWord[12].15 := AlarmSR[12,15].Q1;
hmi_AlarmWord[13].0 := AlarmSR[13,0].Q1;
hmi_AlarmWord[13].1 := AlarmSR[13,1].Q1;
hmi_AlarmWord[13].2 := AlarmSR[13,2].Q1;
hmi_AlarmWord[13].3 := AlarmSR[13,3].Q1;
hmi_AlarmWord[13].4 := AlarmSR[13,4].Q1;
hmi_AlarmWord[13].5 := AlarmSR[13,5].Q1;
hmi_AlarmWord[13].6 := AlarmSR[13,6].Q1;
hmi_AlarmWord[13].7 := AlarmSR[13,7].Q1;
hmi_AlarmWord[13].8 := AlarmSR[13,8].Q1;
hmi_AlarmWord[13].9 := AlarmSR[13,9].Q1;
hmi_AlarmWord[13].10 := AlarmSR[13,10].Q1;
hmi_AlarmWord[13].11 := AlarmSR[13,11].Q1;
hmi_AlarmWord[13].12 := AlarmSR[13,12].Q1;
hmi_AlarmWord[13].13 := AlarmSR[13,13].Q1;
hmi_AlarmWord[13].14 := AlarmSR[13,14].Q1;
hmi_AlarmWord[13].15 := AlarmSR[13,15].Q1;
hmi_AlarmWord[13].0 := AlarmSR[13,0].Q1;
hmi_AlarmWord[13].1 := AlarmSR[13,1].Q1;
hmi_AlarmWord[13].2 := AlarmSR[13,2].Q1;
hmi_AlarmWord[13].3 := AlarmSR[13,3].Q1;
hmi_AlarmWord[13].4 := AlarmSR[13,4].Q1;
hmi_AlarmWord[13].5 := AlarmSR[13,5].Q1;
hmi_AlarmWord[13].6 := AlarmSR[13,6].Q1;
hmi_AlarmWord[13].7 := AlarmSR[13,7].Q1;
hmi_AlarmWord[13].8 := AlarmSR[13,8].Q1;
hmi_AlarmWord[13].9 := AlarmSR[13,9].Q1;
hmi_AlarmWord[13].10 := AlarmSR[13,10].Q1;
hmi_AlarmWord[13].11 := AlarmSR[13,11].Q1;
hmi_AlarmWord[13].12 := AlarmSR[13,12].Q1;
hmi_AlarmWord[13].13 := AlarmSR[13,13].Q1;
hmi_AlarmWord[13].14 := AlarmSR[13,14].Q1;
hmi_AlarmWord[13].15 := AlarmSR[13,15].Q1;
hmi_AlarmWord[14].0 := AlarmSR[14,0].Q1;
hmi_AlarmWord[14].1 := AlarmSR[14,1].Q1;
hmi_AlarmWord[14].2 := AlarmSR[14,2].Q1;
hmi_AlarmWord[14].3 := AlarmSR[14,3].Q1;
hmi_AlarmWord[14].4 := AlarmSR[14,4].Q1;
hmi_AlarmWord[14].5 := AlarmSR[14,5].Q1;
hmi_AlarmWord[14].6 := AlarmSR[14,6].Q1;
hmi_AlarmWord[14].7 := AlarmSR[14,7].Q1;
hmi_AlarmWord[14].8 := AlarmSR[14,8].Q1;
hmi_AlarmWord[14].9 := AlarmSR[14,9].Q1;
hmi_AlarmWord[14].10 := AlarmSR[14,10].Q1;
hmi_AlarmWord[14].11 := AlarmSR[14,11].Q1;
hmi_AlarmWord[14].12 := AlarmSR[14,12].Q1;
hmi_AlarmWord[14].13 := AlarmSR[14,13].Q1;
hmi_AlarmWord[14].14 := AlarmSR[14,14].Q1;
hmi_AlarmWord[14].15 := AlarmSR[14,15].Q1;
hmi_AlarmWord[15].0 := AlarmSR[15,0].Q1;
hmi_AlarmWord[15].1 := AlarmSR[15,1].Q1;
hmi_AlarmWord[15].2 := AlarmSR[15,2].Q1;
hmi_AlarmWord[15].3 := AlarmSR[15,3].Q1;
hmi_AlarmWord[15].4 := AlarmSR[15,4].Q1;
hmi_AlarmWord[15].5 := AlarmSR[15,5].Q1;
hmi_AlarmWord[15].6 := AlarmSR[15,6].Q1;
hmi_AlarmWord[15].7 := AlarmSR[15,7].Q1;
hmi_AlarmWord[15].8 := AlarmSR[15,8].Q1;
hmi_AlarmWord[15].9 := AlarmSR[15,9].Q1;
hmi_AlarmWord[15].10 := AlarmSR[15,10].Q1;
hmi_AlarmWord[15].11 := AlarmSR[15,11].Q1;
hmi_AlarmWord[15].12 := AlarmSR[15,12].Q1;
hmi_AlarmWord[15].13 := AlarmSR[15,13].Q1;
hmi_AlarmWord[15].14 := AlarmSR[15,14].Q1;
hmi_AlarmWord[15].15 := AlarmSR[15,15].Q1;
hmi_AlarmWord[16].0 := AlarmSR[16,0].Q1;
hmi_AlarmWord[16].1 := AlarmSR[16,1].Q1;
hmi_AlarmWord[16].2 := AlarmSR[16,2].Q1;
hmi_AlarmWord[16].3 := AlarmSR[16,3].Q1;
hmi_AlarmWord[16].4 := AlarmSR[16,4].Q1;
hmi_AlarmWord[16].5 := AlarmSR[16,5].Q1;
hmi_AlarmWord[16].6 := AlarmSR[16,6].Q1;
hmi_AlarmWord[16].7 := AlarmSR[16,7].Q1;
hmi_AlarmWord[16].8 := AlarmSR[16,8].Q1;
hmi_AlarmWord[16].9 := AlarmSR[16,9].Q1;
hmi_AlarmWord[16].10 := AlarmSR[16,10].Q1;
hmi_AlarmWord[16].11 := AlarmSR[16,11].Q1;
hmi_AlarmWord[16].12 := AlarmSR[16,12].Q1;
hmi_AlarmWord[16].13 := AlarmSR[16,13].Q1;
hmi_AlarmWord[16].14 := AlarmSR[16,14].Q1;
hmi_AlarmWord[16].15 := AlarmSR[16,15].Q1;
hmi_AlarmWord[17].0 := AlarmSR[17,0].Q1;
hmi_AlarmWord[17].1 := AlarmSR[17,1].Q1;
hmi_AlarmWord[17].2 := AlarmSR[17,2].Q1;
hmi_AlarmWord[17].3 := AlarmSR[17,3].Q1;
hmi_AlarmWord[17].4 := AlarmSR[17,4].Q1;
hmi_AlarmWord[17].5 := AlarmSR[17,5].Q1;
hmi_AlarmWord[17].6 := AlarmSR[17,6].Q1;
hmi_AlarmWord[17].7 := AlarmSR[17,7].Q1;
hmi_AlarmWord[17].8 := AlarmSR[17,8].Q1;
hmi_AlarmWord[17].9 := AlarmSR[17,9].Q1;
hmi_AlarmWord[17].10 := AlarmSR[17,10].Q1;
hmi_AlarmWord[17].11 := AlarmSR[17,11].Q1;
hmi_AlarmWord[17].12 := AlarmSR[17,12].Q1;
hmi_AlarmWord[17].13 := AlarmSR[17,13].Q1;
hmi_AlarmWord[17].14 := AlarmSR[17,14].Q1;
hmi_AlarmWord[17].15 := AlarmSR[17,15].Q1;
hmi_AlarmWord[18].0 := AlarmSR[18,0].Q1;
hmi_AlarmWord[18].1 := AlarmSR[18,1].Q1;
hmi_AlarmWord[18].2 := AlarmSR[18,2].Q1;
hmi_AlarmWord[18].3 := AlarmSR[18,3].Q1;
hmi_AlarmWord[18].4 := AlarmSR[18,4].Q1;
hmi_AlarmWord[18].5 := AlarmSR[18,5].Q1;
hmi_AlarmWord[18].6 := AlarmSR[18,6].Q1;
hmi_AlarmWord[18].7 := AlarmSR[18,7].Q1;
hmi_AlarmWord[18].8 := AlarmSR[18,8].Q1;
hmi_AlarmWord[18].9 := AlarmSR[18,9].Q1;
hmi_AlarmWord[18].10 := AlarmSR[18,10].Q1;
hmi_AlarmWord[18].11 := AlarmSR[18,11].Q1;
hmi_AlarmWord[18].12 := AlarmSR[18,12].Q1;
hmi_AlarmWord[18].13 := AlarmSR[18,13].Q1;
hmi_AlarmWord[18].14 := AlarmSR[18,14].Q1;
hmi_AlarmWord[18].15 := AlarmSR[18,15].Q1;
hmi_AlarmWord[19].0 := AlarmSR[19,0].Q1;
hmi_AlarmWord[19].1 := AlarmSR[19,1].Q1;
hmi_AlarmWord[19].2 := AlarmSR[19,2].Q1;
hmi_AlarmWord[19].3 := AlarmSR[19,3].Q1;
hmi_AlarmWord[19].4 := AlarmSR[19,4].Q1;
hmi_AlarmWord[19].5 := AlarmSR[19,5].Q1;
hmi_AlarmWord[19].6 := AlarmSR[19,6].Q1;
hmi_AlarmWord[19].7 := AlarmSR[19,7].Q1;
hmi_AlarmWord[19].8 := AlarmSR[19,8].Q1;
hmi_AlarmWord[19].9 := AlarmSR[19,9].Q1;
hmi_AlarmWord[19].10 := AlarmSR[19,10].Q1;
hmi_AlarmWord[19].11 := AlarmSR[19,11].Q1;
hmi_AlarmWord[19].12 := AlarmSR[19,12].Q1;
hmi_AlarmWord[19].13 := AlarmSR[19,13].Q1;
hmi_AlarmWord[19].14 := AlarmSR[19,14].Q1;
hmi_AlarmWord[19].15 := AlarmSR[19,15].Q1;

END_ACTION
END_ACTIONS

(* ---- PRG_AO.st ---- *)
PROGRAM PRG_AO
VAR
	BatteryVoltage_pc_minmax_range: 	REAL; 	(*Battery Bus voltage, part of which is over the minimum voltage as defined by sourceminvoltage*)
	BatteryChargeDischargeCurrent_pc: 	REAL;	(*Battery charge or discharge current in percent of sourcenominalcurrent*)
	BatteryVoltage_pc: 					REAL;	(*Battery voltage in percent of range between min and max source voltage*)
	BatteryPower_pc: 					REAL;	(*Battery power in percent of sourcenompower*)
	BatteryCurrent_pc: 					REAL;	(*Battery current in percent of sourcenominalcurrent*)
	BatterySoC_pc:						REAL;	(*Battery State of Charge in percent*)

	BatteryChargeDischargeCurrent_eng: 	REAL;	(*Battery charge or discharge current in Ampere*)
	BatteryVoltage_eng: 				REAL;	(*Battery voltage in volt*)
	BatteryPower_eng: 					REAL;	(*Battery power in kilowatt*)
	BatteryCurrent_eng: 				REAL;	(*Battery current in ampere*)
	BatterySoC_eng:						REAL;	(*Battery State of Charge in kWh*)

	BatteryChargeDischargeCurrent_Instr: 	REAL;	(*Battery charge or discharge current value to instrument*)
	BatteryVoltage_Instr: 					REAL;	(*Battery voltage value to instrument*)
	BatteryPower_Instr: 					REAL;	(*Battery power value to instrument*)
	BatteryCurrent_Instr: 					REAL;	(*Battery current value to instrument*)
	BatterySoC_Instr:						REAL;	(*Battery State of Charge value to instrument*)

	F_Trig : ARRAY[1..cnst_num_ao] OF F_TRIG;
	i : INT;	(*Loop variable*)
	ManualFixChannels : BOOL; (*Will reset channels if faulty, i.e. card number is zero*)
	Reset: BOOL;
	Firstrun : BOOL;

	(*Internal variables*)
	CurrentFilter : 				FILTER_I;
	PowerFilter : 					FILTER_I;
	VoltageFilter : 				FILTER_I;
	ChargeDischargeLimitFilter : 	FILTER_I;
	SoCFilter: 						FILTER_I;

	(*Analog Outputs*)
	ao_BatteryCurrentInstr_daemon: fb_AoProcess;
	ao_BatteryPowerInstr_daemon: fb_AoProcess;
	ao_BatteryVoltageInstr_daemon: fb_AoProcess;
	ao_BatterySocInstr_daemon: fb_AoProcess;
	ao_BatteryChrgDischrgInstr_daemon: fb_AoProcess;

	ao_BatteryCurrentInstr: str_AoProcess;
	ao_BatteryPowerInstr: str_AoProcess;
	ao_BatteryVoltageInstr: str_AoProcess;
	ao_BatterySocInstr: str_AoProcess;
	ao_BatteryChrgDischrgInstr: str_AoProcess;
END_VAR

VAR RETAIN
	ao_BatteryCurrentInstr_setup: str_AoSetup;
	ao_BatteryPowerInstr_setup: str_AoSetup;
	ao_BatteryVoltageInstr_setup: str_AoSetup;
	ao_BatterySocInstr_setup: str_AoSetup;
	ao_BatteryChrgDischrgInstr_setup: str_AoSetup;
END_VAR

Reset := PRG_Functions.Reset;

(*Setup the HMI variables so that they are equal to actual used variables*)
IF (NOT Firstrun) THEN
	hmi_AoSetup[1] := ao_BatteryCurrentInstr_setup;
	hmi_AoSetup[2] := ao_BatteryPowerInstr_setup;
	hmi_AoSetup[3] := ao_BatteryVoltageInstr_setup;
	hmi_AoSetup[4] := ao_BatterySocInstr_setup;
	hmi_AoSetup[5] := ao_BatteryChrgDischrgInstr_setup;
	Firstrun := TRUE;
END_IF

IF PRG_HMI.DoorSettings.enAmpInstrument THEN
	ao_BatteryCurrentInstr_daemon (setup:=ao_BatteryCurrentInstr_setup,reset:=Reset,inPV:=ao_BatteryCurrentInstr);
	hmi_AoPV[1]:=ao_BatteryCurrentInstr_daemon.inPV;
END_IF

IF PRG_HMI.DoorSettings.enkWInstrument THEN
	ao_BatteryPowerInstr_daemon (setup:=ao_BatteryPowerInstr_setup,reset:=Reset,inPV:=ao_BatteryPowerInstr);
	hmi_AoPV[2]:=ao_BatteryPowerInstr_daemon.inPV;
END_IF

IF PRG_HMI.DoorSettings.enVoltInstrument THEN
	ao_BatteryVoltageInstr_daemon (setup:=ao_BatteryVoltageInstr_setup,reset:=Reset,inPV:=ao_BatteryVoltageInstr);
	hmi_AoPV[3]:=ao_BatteryVoltageInstr_daemon.inPV;
END_IF

IF PRG_HMI.DoorSettings.enSoCInstrument THEN
	ao_BatterySocInstr_daemon (setup:=ao_BatterySocInstr_setup,reset:=Reset,inPV:=ao_BatterySocInstr);
	hmi_AoPV[4]:=ao_BatterySocInstr_daemon.inPV;
END_IF

IF PRG_HMI.DoorSettings.enChrgDischrgInstrument THEN
	ao_BatteryChrgDischrgInstr_daemon (setup:=ao_BatteryChrgDischrgInstr_setup,reset:=Reset,inPV:=ao_BatteryChrgDischrgInstr);
	hmi_AoPV[5]:=ao_BatteryChrgDischrgInstr_daemon.inPV;
END_IF

(*---------------------------------------- Channel initialization ----------------------------------------------*)

IF (ManualFixChannels) THEN  (*If manually forced: re-configure the channels*)
	FOR i:=0 TO cnst_num_ao BY 1 DO				(*Check if channel info is empty and restore if so.*)
		IF (hmi_AoSetup[i].CardNb = 0 AND PRG_HMI.setup_AioCard1_Number <> 0) THEN
			hmi_RestoreDefault_ao[i] := TRUE;
		END_IF
	END_FOR;
	ManualFixChannels := FALSE;
END_IF

(*
 * =======================================================================================================================================
 * Calculate instrument values in percent (_pc) and engineering values (_eng)
 * =======================================================================================================================================
*)

BatteryCurrent_pc := 100*fun_SafeDivide(
 						divident := DINT_TO_REAL(ABS(PRG_BatteryComm.CorvusRead[PRG_BatteryComm.M].theArray.busCurrent)) ,
 						devisor := PRG_HMI.DriveSettings.SourceNomCurrent
);
BatteryCurrent_eng := DINT_TO_REAL(PRG_BatteryComm.CorvusRead[PRG_BatteryComm.M].theArray.busCurrent);

BatteryPower_pc := 100*fun_SafeDivide(
 						divident := PRG_BatteryComm.CorvusRead[PRG_BatteryComm.M].theArray.busPowerCalculated ,
 						devisor := PRG_HMI.DriveSettings.SourceNomPower
);
BatteryPower_eng := PRG_BatteryComm.CorvusRead[PRG_BatteryComm.M].theArray.busPowerCalculated;

BatteryVoltage_pc := 100*fun_SafeDivide(
	 						divident :=(PRG_BatteryComm.CorvusRead[PRG_BatteryComm.M].theArray.busVoltage - PRG_HMI.DriveSettings.SourceMinVoltage),
	 						devisor := (PRG_HMI.DriveSettings.SourceMaxVoltage-PRG_HMI.DriveSettings.SourceMinVoltage)
);
BatteryVoltage_eng := PRG_BatteryComm.CorvusRead[PRG_BatteryComm.M].theArray.busVoltage;

BatterySoC_pc := PRG_BatteryComm.CorvusRead[PRG_BatteryComm.M].theArray.systemOnlineSOC;
BatterySoC_eng := PRG_Battery.AvailableEnergy;

IF (PRG_Battery.batteryCharging) THEN
	BatteryChargeDischargeCurrent_pc := 100 * fun_SafeDivide(
 						divident := PRG_Battery.DriveChargeLimit_eng,
 						devisor := PRG_HMI.DriveSettings.SourceNomCurrent
 	);
	BatteryChargeDischargeCurrent_eng := PRG_Battery.DriveChargeLimit_eng;
ELSE
	BatteryChargeDischargeCurrent_pc := 100 * fun_SafeDivide(
 						divident := PRG_Battery.DriveDischargeLimit_eng,
 						devisor := PRG_HMI.DriveSettings.SourceNomCurrent
);
	BatteryChargeDischargeCurrent_eng := PRG_Battery.DriveDischargeLimit_eng;
END_IF

(*
 * =======================================================================================================================================
 * Select percent (_pc) or engineering values (_eng)
 * =======================================================================================================================================
*)
IF (PRG_HMI.DoorSettings.enPercentAmpInstrument) THEN
	BatteryCurrent_Instr :=  BatteryCurrent_pc;
ELSE
	BatteryCurrent_Instr := BatteryCurrent_eng;
END_IF

IF (PRG_HMI.DoorSettings.enPercentVoltInstrument) THEN
	BatteryVoltage_Instr :=  BatteryVoltage_pc;
ELSE
	BatteryVoltage_Instr := BatteryVoltage_eng;
END_IF

IF (PRG_HMI.DoorSettings.enPercentkWInstrument) THEN
	BatteryPower_Instr :=  BatteryPower_pc;
ELSE
	BatteryPower_Instr := BatteryPower_eng;
END_IF

IF (PRG_HMI.DoorSettings.enPercentSoCInstrument) THEN
	BatterySoC_Instr :=  BatterySoC_pc;
ELSE
	BatterySoC_Instr := BatterySoC_eng;
END_IF

IF (PRG_HMI.DoorSettings.enPercentChrgDischrgInstrument) THEN
	BatteryChargeDischargeCurrent_Instr :=  BatteryChargeDischargeCurrent_pc;
ELSE
	BatteryChargeDischargeCurrent_Instr := BatteryChargeDischargeCurrent_eng;
END_IF

(*
 * =======================================================================================================================================
 * Enable absolute values
 * =======================================================================================================================================
*)
IF (PRG_HMI.DoorSettings.enAbsValuesAmpInstrument) THEN
	BatteryCurrent_Instr :=  ABS(BatteryCurrent_Instr);
END_IF

IF (PRG_HMI.DoorSettings.enAbsValuesVoltInstrument) THEN
	BatteryVoltage_Instr :=  ABS(BatteryVoltage_Instr);
END_IF

IF (PRG_HMI.DoorSettings.enAbsValueskWInstrument) THEN
	BatteryPower_Instr :=  ABS(BatteryPower_Instr);
END_IF

IF (PRG_HMI.DoorSettings.enAbsValuesSoCInstrument) THEN
	BatterySoC_Instr :=  ABS(BatterySoC_Instr);
END_IF

IF (PRG_HMI.DoorSettings.enAbsValuesChrgDischrgInstrument) THEN
	BatteryChargeDischargeCurrent_Instr :=  ABS(BatteryChargeDischargeCurrent_Instr);
END_IF

(*
 * =======================================================================================================================================
 * Filter outputs
 * =======================================================================================================================================
*)

CurrentFilter(
	X := REAL_TO_INT(BatteryCurrent_Instr),
	T := PRG_HMI.DoorSettings.InstrumentFilterTime,
	Y => ao_BatteryCurrentInstr.PV
);

VoltageFilter(
	X := REAL_TO_INT(BatteryVoltage_Instr),
	T := PRG_HMI.DoorSettings.InstrumentFilterTime,
	Y => ao_BatteryVoltageInstr.PV
);

PowerFilter(
	X := REAL_TO_INT(BatteryPower_Instr),
	T := PRG_HMI.DoorSettings.InstrumentFilterTime,
	Y => ao_BatteryPowerInstr.PV
);

ChargeDischargeLimitFilter(
	X := LIMIT(0, REAL_TO_INT(BatteryChargeDischargeCurrent_pc), REAL_TO_INT(PRG_HMI.DriveSettings.SourceNomCurrent)),
	T := PRG_HMI.DoorSettings.InstrumentFilterTime,
	Y => ao_BatteryChrgDischrgInstr.PV
);

SoCFilter(
	X := REAL_TO_INT(BatterySoC_Instr),
	T := PRG_HMI.DoorSettings.InstrumentFilterTime,
	Y => ao_BatterySocInstr.PV
);

ChargeDischargeLimitFilter(
	X := REAL_TO_INT(BatteryChargeDischargeCurrent_Instr),
	T := PRG_HMI.DoorSettings.InstrumentFilterTime,
	Y => ao_BatteryChrgDischrgInstr.PV
);

END_PROGRAM

ACTIONS

ACTION Settings

(***************ao_BatteryCurrentInstr***************)
IF (RestoreAllToDefault OR ao_BatteryCurrentInstr_setup.RestoreDefault  OR hmi_RestoreDefault_ao[1]) THEN
	ao_BatteryCurrentInstr_setup.Name:='ao_BatteryCurrentInstr';
	ao_BatteryCurrentInstr_setup.CardNb:=PRG_HMI.setup_AioCard1_Number;
	ao_BatteryCurrentInstr_setup.ChannelMode:=16#62;
	ao_BatteryCurrentInstr_setup.ChannelNb:=3;
 	ao_BatteryCurrentInstr_setup.Enable.Forcing:=0;
 	ao_BatteryCurrentInstr_setup.Enable.WireBreak:=1;
 	ao_BatteryCurrentInstr_setup.Enable.OOR:=1;
 	ao_BatteryCurrentInstr_setup.Delay.WireBreak:=T#1s;
 	ao_BatteryCurrentInstr_setup.Delay.OoR:=T#1s;
 	ao_BatteryCurrentInstr_setup.Levels.minPv:=0;
 	ao_BatteryCurrentInstr_setup.Levels.maxPv:=120;
 	ao_BatteryCurrentInstr_setup.Levels.MinOutputRaw:=0;
 	ao_BatteryCurrentInstr_setup.Levels.MaxOutputRaw:=65536;
 	ao_BatteryCurrentInstr_setup.Levels.ForceValue:=0;
END_IF
IF (hmi_RestoreDefault_ao[1] OR RestoreAllToDefault OR ao_BatteryCurrentInstr_setup.RestoreDefault) THEN (*Copy values into HMI variable and reset*)
	hmi_AoSetup[1]:=ao_BatteryCurrentInstr_setup; (*Copy setup values from retain into hmi variable*)
	hmi_RestoreDefault_ao[1]:=FALSE; (*Make sure that the restore variable is turned off after one restore command*)
	ao_BatteryCurrentInstr_setup.RestoreDefault:=FALSE; (*Make sure that the restore variable is turned off after one restore command*)
END_IF
IF (hmi_AoWriteSetup[1]) THEN
	ao_BatteryCurrentInstr_setup:=hmi_AoSetup[1]; (*Paste hmi changes back into setup variable*)
	hmi_AoWriteSetup[1]:=FALSE; (*Make sure that the write variable is turned off after one write command*)
END_IF
F_Trig[1](CLK:=hmi_AoPV[1].IsForced); (*Reset HMI forcing dialog when timer runs out*)
IF (F_Trig[1].Q) THEN hmi_AoSetup[1].Enable.Forcing:=FALSE;ao_BatteryCurrentInstr_setup.Enable.Forcing:=FALSE; END_IF
(**************************************************)

(***************ao_BatteryPowerInstr***************)
IF (RestoreAllToDefault OR ao_BatteryPowerInstr_setup.RestoreDefault  OR hmi_RestoreDefault_ao[2]) THEN
	ao_BatteryPowerInstr_setup.Name:='ao_BatteryPowerInstr';
	ao_BatteryPowerInstr_setup.CardNb:=PRG_HMI.setup_AioCard1_Number;
	ao_BatteryPowerInstr_setup.ChannelMode:=16#62;
	ao_BatteryPowerInstr_setup.ChannelNb:=5;
 	ao_BatteryPowerInstr_setup.Enable.Forcing:=0;
 	ao_BatteryPowerInstr_setup.Enable.WireBreak:=1;
 	ao_BatteryPowerInstr_setup.Enable.OOR:=1;
 	ao_BatteryPowerInstr_setup.Delay.WireBreak:=T#1s;
 	ao_BatteryPowerInstr_setup.Delay.OoR:=T#1s;
 	ao_BatteryPowerInstr_setup.Levels.minPv:=0;
 	ao_BatteryPowerInstr_setup.Levels.maxPv:=120;
 	ao_BatteryPowerInstr_setup.Levels.MinOutputRaw:=0;
 	ao_BatteryPowerInstr_setup.Levels.MaxOutputRaw:=65536;
 	ao_BatteryPowerInstr_setup.Levels.ForceValue:=0;
END_IF
IF (hmi_RestoreDefault_ao[2] OR RestoreAllToDefault OR ao_BatteryPowerInstr_setup.RestoreDefault) THEN (*Copy values into HMI variable and reset*)
	hmi_AoSetup[2]:=ao_BatteryPowerInstr_setup; (*Copy setup values from retain into hmi variable*)
	hmi_RestoreDefault_ao[2]:=FALSE; (*Make sure that the restore variable is turned off after one restore command*)
	ao_BatteryPowerInstr_setup.RestoreDefault:=FALSE; (*Make sure that the restore variable is turned off after one restore command*)
END_IF
IF (hmi_AoWriteSetup[2]) THEN
	ao_BatteryPowerInstr_setup:=hmi_AoSetup[2]; (*Paste hmi changes back into setup variable*)
	hmi_AoWriteSetup[2]:=FALSE; (*Make sure that the write variable is turned off after one write command*)
END_IF
F_Trig[2](CLK:=hmi_AoPV[2].IsForced); (*Reset HMI forcing dialog when timer runs out*)
IF (F_Trig[2].Q) THEN hmi_AoSetup[2].Enable.Forcing:=FALSE;ao_BatteryPowerInstr_setup.Enable.Forcing:=FALSE; END_IF
(**************************************************)

(***************ao_BatteryVoltageInstr***************)
IF (RestoreAllToDefault OR ao_BatteryVoltageInstr_setup.RestoreDefault  OR hmi_RestoreDefault_ao[3]) THEN
	ao_BatteryVoltageInstr_setup.Name:='ao_BatteryVoltageInstr';
	ao_BatteryVoltageInstr_setup.CardNb:=PRG_HMI.setup_AioCard1_Number;
	ao_BatteryVoltageInstr_setup.ChannelMode:=16#62;
	ao_BatteryVoltageInstr_setup.ChannelNb:=7;
 	ao_BatteryVoltageInstr_setup.Enable.Forcing:=0;
 	ao_BatteryVoltageInstr_setup.Enable.WireBreak:=1;
 	ao_BatteryVoltageInstr_setup.Enable.OOR:=1;
 	ao_BatteryVoltageInstr_setup.Delay.WireBreak:=T#1s;
 	ao_BatteryVoltageInstr_setup.Delay.OoR:=T#1s;
 	ao_BatteryVoltageInstr_setup.Levels.minPv:=0;
 	ao_BatteryVoltageInstr_setup.Levels.maxPv:=120;
 	ao_BatteryVoltageInstr_setup.Levels.MinOutputRaw:=0;
 	ao_BatteryVoltageInstr_setup.Levels.MaxOutputRaw:=65536;
 	ao_BatteryVoltageInstr_setup.Levels.ForceValue:=0;
END_IF
IF (hmi_RestoreDefault_ao[3] OR RestoreAllToDefault OR ao_BatteryVoltageInstr_setup.RestoreDefault) THEN (*Copy values into HMI variable and reset*)
	hmi_AoSetup[3]:=ao_BatteryVoltageInstr_setup; (*Copy setup values from retain into hmi variable*)
	hmi_RestoreDefault_ao[3]:=FALSE; (*Make sure that the restore variable is turned off after one restore command*)
	ao_BatteryVoltageInstr_setup.RestoreDefault:=FALSE; (*Make sure that the restore variable is turned off after one restore command*)
END_IF
IF (hmi_AoWriteSetup[3]) THEN
	ao_BatteryVoltageInstr_setup:=hmi_AoSetup[3]; (*Paste hmi changes back into setup variable*)
	hmi_AoWriteSetup[3]:=FALSE; (*Make sure that the write variable is turned off after one write command*)
END_IF
F_Trig[3](CLK:=hmi_AoPV[3].IsForced); (*Reset HMI forcing dialog when timer runs out*)
IF (F_Trig[3].Q) THEN hmi_AoSetup[3].Enable.Forcing:=FALSE;ao_BatteryVoltageInstr_setup.Enable.Forcing:=FALSE; END_IF
(**************************************************)

(***************ao_BatterySocInstr***************)
IF (RestoreAllToDefault OR ao_BatterySocInstr_setup.RestoreDefault  OR hmi_RestoreDefault_ao[4]) THEN
	ao_BatterySocInstr_setup.Name:='ao_BatterySocInstr';
	ao_BatterySocInstr_setup.CardNb:=PRG_HMI.setup_AioCard1_Number;
	ao_BatterySocInstr_setup.ChannelMode:=16#62;
	ao_BatterySocInstr_setup.ChannelNb:=9;
 	ao_BatterySocInstr_setup.Enable.Forcing:=0;
 	ao_BatterySocInstr_setup.Enable.WireBreak:=1;
 	ao_BatterySocInstr_setup.Enable.OOR:=1;
 	ao_BatterySocInstr_setup.Delay.WireBreak:=T#1s;
 	ao_BatterySocInstr_setup.Delay.OoR:=T#1s;
 	ao_BatterySocInstr_setup.Levels.minPv:=0;
 	ao_BatterySocInstr_setup.Levels.maxPv:=120;
 	ao_BatterySocInstr_setup.Levels.MinOutputRaw:=0;
 	ao_BatterySocInstr_setup.Levels.MaxOutputRaw:=65536;
 	ao_BatterySocInstr_setup.Levels.ForceValue:=0;
END_IF
IF (hmi_RestoreDefault_ao[4] OR RestoreAllToDefault OR ao_BatterySocInstr_setup.RestoreDefault) THEN (*Copy values into HMI variable and reset*)
	hmi_AoSetup[4]:=ao_BatterySocInstr_setup; (*Copy setup values from retain into hmi variable*)
	hmi_RestoreDefault_ao[4]:=FALSE; (*Make sure that the restore variable is turned off after one restore command*)
	ao_BatterySocInstr_setup.RestoreDefault:=FALSE; (*Make sure that the restore variable is turned off after one restore command*)
END_IF
IF (hmi_AoWriteSetup[4]) THEN
	ao_BatterySocInstr_setup:=hmi_AoSetup[4]; (*Paste hmi changes back into setup variable*)
	hmi_AoWriteSetup[4]:=FALSE; (*Make sure that the write variable is turned off after one write command*)
END_IF
F_Trig[4](CLK:=hmi_AoPV[4].IsForced); (*Reset HMI forcing dialog when timer runs out*)
IF (F_Trig[4].Q) THEN hmi_AoSetup[4].Enable.Forcing:=FALSE;ao_BatterySocInstr_setup.Enable.Forcing:=FALSE; END_IF
(**************************************************)

(***************ao_BatteryChrgDischrgInstr***************)
IF (RestoreAllToDefault OR ao_BatteryChrgDischrgInstr_setup.RestoreDefault  OR hmi_RestoreDefault_ao[5]) THEN
	ao_BatteryChrgDischrgInstr_setup.Name:='ao_BatteryChrgDischrgInstr';
	ao_BatteryChrgDischrgInstr_setup.CardNb:=PRG_HMI.setup_AioCard1_Number;
	ao_BatteryChrgDischrgInstr_setup.ChannelMode:=16#62;
	ao_BatteryChrgDischrgInstr_setup.ChannelNb:=11;
 	ao_BatteryChrgDischrgInstr_setup.Enable.Forcing:=0;
 	ao_BatteryChrgDischrgInstr_setup.Enable.WireBreak:=1;
 	ao_BatteryChrgDischrgInstr_setup.Enable.OOR:=1;
 	ao_BatteryChrgDischrgInstr_setup.Delay.WireBreak:=T#1s;
 	ao_BatteryChrgDischrgInstr_setup.Delay.OoR:=T#1s;
 	ao_BatteryChrgDischrgInstr_setup.Levels.minPv:=0;
 	ao_BatteryChrgDischrgInstr_setup.Levels.maxPv:=120;
 	ao_BatteryChrgDischrgInstr_setup.Levels.MinOutputRaw:=0;
 	ao_BatteryChrgDischrgInstr_setup.Levels.MaxOutputRaw:=65536;
 	ao_BatteryChrgDischrgInstr_setup.Levels.ForceValue:=0;
END_IF
IF (hmi_RestoreDefault_ao[5] OR RestoreAllToDefault OR ao_BatteryChrgDischrgInstr_setup.RestoreDefault) THEN (*Copy values into HMI variable and reset*)
	hmi_AoSetup[5]:=ao_BatteryChrgDischrgInstr_setup; (*Copy setup values from retain into hmi variable*)
	hmi_RestoreDefault_ao[5]:=FALSE; (*Make sure that the restore variable is turned off after one restore command*)
	ao_BatteryChrgDischrgInstr_setup.RestoreDefault:=FALSE; (*Make sure that the restore variable is turned off after one restore command*)
END_IF
IF (hmi_AoWriteSetup[5]) THEN
	ao_BatteryChrgDischrgInstr_setup:=hmi_AoSetup[5]; (*Paste hmi changes back into setup variable*)
	hmi_AoWriteSetup[5]:=FALSE; (*Make sure that the write variable is turned off after one write command*)
END_IF
F_Trig[5](CLK:=hmi_AoPV[5].IsForced); (*Reset HMI forcing dialog when timer runs out*)
IF (F_Trig[5].Q) THEN hmi_AoSetup[5].Enable.Forcing:=FALSE;ao_BatteryChrgDischrgInstr_setup.Enable.Forcing:=FALSE; END_IF
(**************************************************)

END_ACTION

END_ACTIONS

(* ---- PRG_DI.st ---- *)
PROGRAM PRG_DI
VAR
	F_Trig : ARRAY[1..cnst_num_di] OF F_TRIG;
	i : INT;
	ManualFixChannels : BOOL; (*Will reset channels if faulty, i.e. card number is zero*)
	Reset: BOOL;
	Firstrun : BOOL;

	di_DcBreakerEarlyBreak_daemon: fb_DiProcess;
	di_LocalIncrease_daemon: fb_DiProcess;
	di_LocalDecrease_daemon: fb_DiProcess;
	di_LocalMode_daemon: fb_DiProcess;
	di_RemoteMode_daemon: fb_DiProcess;
	di_LocalStart_daemon: fb_DiProcess;
	di_LocalStop_daemon: fb_DiProcess;
	di_LocalReset_daemon: fb_DiProcess;
	di_LocalEmergencyStop_daemon: fb_DiProcess;
	di_FusesOK_daemon: fb_DiProcess;
	di_DcBreakerOpen_daemon: fb_DiProcess;
	di_DcBreakerClosed_daemon: fb_DiProcess;
	di_EthernetSwitchAlarm_daemon: fb_DiProcess;
	di_EmergencyStopLoopFault_daemon: fb_DiProcess;
	di_BatteryAuxOK_daemon: fb_DiProcess;
	di_BatteryAuxNotOK_daemon: fb_DiProcess;
	di_WaterLeakageDetected_daemon: fb_DiProcess;
	di_RemoteEmergencyStop_daemon: fb_DiProcess;
	di_SpareChannel32_daemon: fb_DiProcess;

	di_DcBreakerEarlyBreak: str_DiProcess;
	di_LocalIncrease: str_DiProcess;
	di_LocalDecrease: str_DiProcess;
	di_LocalMode: str_DiProcess;
	di_RemoteMode: str_DiProcess;
	di_LocalStart: str_DiProcess;
	di_LocalStop: str_DiProcess;
	di_LocalReset: str_DiProcess;
	di_LocalEmergencyStop: str_DiProcess;
	di_FusesOK: str_DiProcess;
	di_DcBreakerOpen: str_DiProcess;
	di_DcBreakerClosed: str_DiProcess;
	di_EthernetSwitchAlarm: str_DiProcess;
	di_EmergencyStopLoopFault: str_DiProcess;
	di_BatteryAuxOK: str_DiProcess;
	di_BatteryAuxNotOK: str_DiProcess;
	di_WaterLeakageDetected: str_DiProcess;
	di_RemoteEmergencyStop: str_DiProcess;
	di_SpareChannel32: str_DiProcess;
END_VAR

VAR RETAIN
	di_DcBreakerEarlyBreak_setup: str_DiSetup;
	di_LocalIncrease_setup: str_DiSetup;
	di_LocalDecrease_setup: str_DiSetup;
	di_LocalMode_setup: str_DiSetup;
	di_RemoteMode_setup: str_DiSetup;
	di_LocalStart_setup: str_DiSetup;
	di_LocalStop_setup: str_DiSetup;
	di_LocalReset_setup: str_DiSetup;
	di_LocalEmergencyStop_setup: str_DiSetup;
	di_FusesOK_setup: str_DiSetup;
	di_DcBreakerOpen_setup: str_DiSetup;
	di_DcBreakerClosed_setup: str_DiSetup;
	di_EthernetSwitchAlarm_setup: str_DiSetup;
	di_EmergencyStopLoopFault_setup: str_DiSetup;
	di_BatteryAuxOK_setup: str_DiSetup;
	di_BatteryAuxNotOK_setup: str_DiSetup;
	di_WaterLeakageDetected_setup: str_DiSetup;
	di_RemoteEmergencyStop_setup: str_DiSetup;
	di_SpareChannel32_setup: str_DiSetup;
END_VAR

Reset := PRG_Functions.Reset;

(*Setup the HMI variables so that they are equal to actual used variables*)
IF (NOT Firstrun) THEN
	hmi_DiSetup[1]:=di_DcBreakerEarlyBreak_setup;
	hmi_DiSetup[2]:=di_LocalIncrease_setup;
	hmi_DiSetup[3]:=di_LocalDecrease_setup;
	hmi_DiSetup[4]:=di_LocalMode_setup;
	hmi_DiSetup[5]:=di_RemoteMode_setup;
	hmi_DiSetup[6]:=di_LocalStart_setup;
	hmi_DiSetup[7]:=di_LocalStop_setup;
	hmi_DiSetup[8]:=di_LocalReset_setup;
	hmi_DiSetup[9]:=di_LocalEmergencyStop_setup;
	hmi_DiSetup[10]:=di_FusesOK_setup;
	hmi_DiSetup[11]:=di_DcBreakerOpen_setup;
	hmi_DiSetup[12]:=di_DcBreakerClosed_setup;
	hmi_DiSetup[13]:=di_EthernetSwitchAlarm_setup;
	hmi_DiSetup[14]:=di_EmergencyStopLoopFault_setup;
	hmi_DiSetup[15]:=di_BatteryAuxOK_setup;
	hmi_DiSetup[16]:=di_BatteryAuxNotOK_setup;
	hmi_DiSetup[17]:=di_WaterLeakageDetected_setup;
	hmi_DiSetup[18]:=di_RemoteEmergencyStop_setup;
	hmi_DiSetup[19]:=di_SpareChannel32_setup;
	Firstrun := TRUE;
END_IF

di_DcBreakerEarlyBreak_daemon (setup:=di_DcBreakerEarlyBreak_setup,outPV=>di_DcBreakerEarlyBreak);
di_LocalIncrease_daemon (setup:=di_LocalIncrease_setup,outPV=>di_LocalIncrease);
di_LocalDecrease_daemon (setup:=di_LocalDecrease_setup,outPV=>di_LocalDecrease);
di_LocalMode_daemon (setup:=di_LocalMode_setup,outPV=>di_LocalMode);
di_RemoteMode_daemon (setup:=di_RemoteMode_setup,outPV=>di_RemoteMode);
di_LocalStart_daemon (setup:=di_LocalStart_setup,outPV=>di_LocalStart);
di_LocalStop_daemon (setup:=di_LocalStop_setup,outPV=>di_LocalStop);
di_LocalReset_daemon (setup:=di_LocalReset_setup,outPV=>di_LocalReset);
di_LocalEmergencyStop_daemon (setup:=di_LocalEmergencyStop_setup,outPV=>di_LocalEmergencyStop);
di_FusesOK_daemon (setup:=di_FusesOK_setup,outPV=>di_FusesOK);
di_DcBreakerOpen_daemon (setup:=di_DcBreakerOpen_setup,outPV=>di_DcBreakerOpen);
di_DcBreakerClosed_daemon (setup:=di_DcBreakerClosed_setup,outPV=>di_DcBreakerClosed);
di_EthernetSwitchAlarm_daemon (setup:=di_EthernetSwitchAlarm_setup,outPV=>di_EthernetSwitchAlarm);
di_EmergencyStopLoopFault_daemon (setup:=di_EmergencyStopLoopFault_setup,outPV=>di_EmergencyStopLoopFault);
di_BatteryAuxOK_daemon (setup:=di_BatteryAuxOK_setup,outPV=>di_BatteryAuxOK);
di_BatteryAuxNotOK_daemon (setup:=di_BatteryAuxNotOK_setup,outPV=>di_BatteryAuxNotOK);
di_WaterLeakageDetected_daemon (setup:=di_WaterLeakageDetected_setup,outPV=>di_WaterLeakageDetected);
di_RemoteEmergencyStop_daemon (setup:=di_RemoteEmergencyStop_setup,outPV=>di_RemoteEmergencyStop);
di_SpareChannel32_daemon (setup:=di_SpareChannel32_setup,outPV=>di_SpareChannel32);

hmi_DiPV[1]:=di_DcBreakerEarlyBreak_daemon.outPV;
hmi_DiPV[2]:=di_LocalIncrease_daemon.outPV;
hmi_DiPV[3]:=di_LocalDecrease_daemon.outPV;
hmi_DiPV[4]:=di_LocalMode_daemon.outPV;
hmi_DiPV[5]:=di_RemoteMode_daemon.outPV;
hmi_DiPV[6]:=di_LocalStart_daemon.outPV;
hmi_DiPV[7]:=di_LocalStop_daemon.outPV;
hmi_DiPV[8]:=di_LocalReset_daemon.outPV;
hmi_DiPV[9]:=di_LocalEmergencyStop_daemon.outPV;
hmi_DiPV[10]:=di_FusesOK_daemon.outPV;
hmi_DiPV[11]:=di_DcBreakerOpen_daemon.outPV;
hmi_DiPV[12]:=di_DcBreakerClosed_daemon.outPV;
hmi_DiPV[13]:=di_EthernetSwitchAlarm_daemon.outPV;
hmi_DiPV[14]:=di_EmergencyStopLoopFault_daemon.outPV;
hmi_DiPV[15]:=di_BatteryAuxOK_daemon.outPV;
hmi_DiPV[16]:=di_BatteryAuxNotOK_daemon.outPV;
hmi_DiPV[17]:=di_WaterLeakageDetected_daemon.outPV;
hmi_DiPV[18]:=di_RemoteEmergencyStop_daemon.outPV;
hmi_DiPV[19]:=di_SpareChannel32_daemon.outPV;

IF (ManualFixChannels) THEN  (*If manually forced: re-configure the channels*)
	FOR i:=1 TO cnst_num_di BY 1 DO			(*Check if channel info is empty and restore if so.*)
		IF (hmi_DiSetup[i].CardNb = 0 AND PRG_HMI.setup_DioCard1_Number <> 0) THEN
			hmi_RestoreDefault_di[i] := TRUE;
		END_IF
	END_FOR;
	ManualFixChannels := FALSE;
END_IF

END_PROGRAM

ACTIONS

ACTION Settings

(**************di_DcBreakerEarlyBreak***********************)
IF (RestoreAllToDefault OR di_DcBreakerEarlyBreak_setup.RestoreDefault  OR hmi_RestoreDefault_di[1]) THEN
	di_DcBreakerEarlyBreak_setup.Name:='di_DcBreakerEarlyBreak';
	di_DcBreakerEarlyBreak_setup.CardNb:=PRG_HMI.setup_DioCard1_Number;
	di_DcBreakerEarlyBreak_setup.ChannelMode:=1;
	di_DcBreakerEarlyBreak_setup.ChannelNb:=7;
 	di_DcBreakerEarlyBreak_setup.Delay.TOF:=T#0ms;
	di_DcBreakerEarlyBreak_setup.Delay.TON:=T#0ms;
	di_DcBreakerEarlyBreak_setup.Enable.Forcing:=0;
	di_DcBreakerEarlyBreak_setup.Enable.TON:=0;
	di_DcBreakerEarlyBreak_setup.Enable.TOF:=0;
	di_DcBreakerEarlyBreak_setup.Levels.ForceValue:=0;
END_IF
IF (hmi_RestoreDefault_di[1] OR RestoreAllToDefault OR di_DcBreakerEarlyBreak_setup.RestoreDefault) THEN (*Copy values into HMI variable and reset*)
	hmi_DiSetup[1]:=di_DcBreakerEarlyBreak_setup; (*Copy setup values from retain into hmi variable*)
	hmi_RestoreDefault_di[1]:=FALSE; (*Make sure that the restore variable is turned off after one restore command*)
	di_DcBreakerEarlyBreak_setup.RestoreDefault:=FALSE; (*Make sure that the restore variable is turned off after one restore command*)
END_IF
IF (hmi_DiWriteSetup[1]) THEN
	di_DcBreakerEarlyBreak_setup:=hmi_DiSetup[1]; (*Paste hmi changes back into setup variable*)
	hmi_DiWriteSetup[1]:=FALSE; (*Make sure that the write variable is turned off after one write command*)
END_IF
F_Trig[1](CLK:=hmi_DiPV[1].IsForced); (*Reset HMI forcing dialog when timer runs out*)
IF (F_Trig[1].Q) THEN hmi_DiSetup[1].Enable.Forcing:=FALSE;di_DcBreakerEarlyBreak_setup.Enable.Forcing:=FALSE; END_IF
(**************************************************)

(**************di_LocalIncrease***********************)
IF (RestoreAllToDefault OR di_LocalIncrease_setup.RestoreDefault  OR hmi_RestoreDefault_di[2]) THEN
	di_LocalIncrease_setup.Name:='di_LocalIncrease';
	di_LocalIncrease_setup.CardNb:=PRG_HMI.setup_DioCard1_Number;
	di_LocalIncrease_setup.ChannelMode:=1;
	di_LocalIncrease_setup.ChannelNb:=8;
 	di_LocalIncrease_setup.Delay.TOF:=T#0ms;
	di_LocalIncrease_setup.Delay.TON:=T#0ms;
	di_LocalIncrease_setup.Enable.Forcing:=0;
	di_LocalIncrease_setup.Enable.TON:=0;
	di_LocalIncrease_setup.Enable.TOF:=0;
	di_LocalIncrease_setup.Levels.ForceValue:=0;
END_IF
IF (hmi_RestoreDefault_di[2] OR RestoreAllToDefault OR di_LocalIncrease_setup.RestoreDefault) THEN (*Copy values into HMI variable and reset*)
	hmi_DiSetup[2]:=di_LocalIncrease_setup; (*Copy setup values from retain into hmi variable*)
	hmi_RestoreDefault_di[2]:=FALSE; (*Make sure that the restore variable is turned off after one restore command*)
	di_LocalIncrease_setup.RestoreDefault:=FALSE; (*Make sure that the restore variable is turned off after one restore command*)
END_IF
IF (hmi_DiWriteSetup[2]) THEN
	di_LocalIncrease_setup:=hmi_DiSetup[2]; (*Paste hmi changes back into setup variable*)
	hmi_DiWriteSetup[2]:=FALSE; (*Make sure that the write variable is turned off after one write command*)
END_IF
F_Trig[2](CLK:=hmi_DiPV[2].IsForced); (*Reset HMI forcing dialog when timer runs out*)
IF (F_Trig[2].Q) THEN hmi_DiSetup[2].Enable.Forcing:=FALSE;di_LocalIncrease_setup.Enable.Forcing:=FALSE; END_IF
(**************************************************)

(**************di_LocalDecrease***********************)
IF (RestoreAllToDefault OR di_LocalDecrease_setup.RestoreDefault  OR hmi_RestoreDefault_di[3]) THEN
	di_LocalDecrease_setup.Name:='di_LocalDecrease';
	di_LocalDecrease_setup.CardNb:=PRG_HMI.setup_DioCard1_Number;
	di_LocalDecrease_setup.ChannelMode:=1;
	di_LocalDecrease_setup.ChannelNb:=9;
 	di_LocalDecrease_setup.Delay.TOF:=T#0ms;
	di_LocalDecrease_setup.Delay.TON:=T#0ms;
	di_LocalDecrease_setup.Enable.Forcing:=0;
	di_LocalDecrease_setup.Enable.TON:=0;
	di_LocalDecrease_setup.Enable.TOF:=0;
	di_LocalDecrease_setup.Levels.ForceValue:=0;
END_IF
IF (hmi_RestoreDefault_di[3] OR RestoreAllToDefault OR di_LocalDecrease_setup.RestoreDefault) THEN (*Copy values into HMI variable and reset*)
	hmi_DiSetup[3]:=di_LocalDecrease_setup; (*Copy setup values from retain into hmi variable*)
	hmi_RestoreDefault_di[3]:=FALSE; (*Make sure that the restore variable is turned off after one restore command*)
	di_LocalDecrease_setup.RestoreDefault:=FALSE; (*Make sure that the restore variable is turned off after one restore command*)
END_IF
IF (hmi_DiWriteSetup[3]) THEN
	di_LocalDecrease_setup:=hmi_DiSetup[3]; (*Paste hmi changes back into setup variable*)
	hmi_DiWriteSetup[3]:=FALSE; (*Make sure that the write variable is turned off after one write command*)
END_IF
F_Trig[3](CLK:=hmi_DiPV[3].IsForced); (*Reset HMI forcing dialog when timer runs out*)
IF (F_Trig[3].Q) THEN hmi_DiSetup[3].Enable.Forcing:=FALSE;di_LocalDecrease_setup.Enable.Forcing:=FALSE; END_IF
(**************************************************)

(**************di_LocalMode***********************)
IF (RestoreAllToDefault OR di_LocalMode_setup.RestoreDefault  OR hmi_RestoreDefault_di[4]) THEN
	di_LocalMode_setup.Name:='di_LocalMode';
	di_LocalMode_setup.CardNb:=PRG_HMI.setup_DioCard1_Number;
	di_LocalMode_setup.ChannelMode:=1;
	di_LocalMode_setup.ChannelNb:=17;
 	di_LocalMode_setup.Delay.TOF:=T#0ms;
	di_LocalMode_setup.Delay.TON:=T#0ms;
	di_LocalMode_setup.Enable.Forcing:=0;
	di_LocalMode_setup.Enable.TON:=0;
	di_LocalMode_setup.Enable.TOF:=0;
	di_LocalMode_setup.Levels.ForceValue:=0;
END_IF
IF (hmi_RestoreDefault_di[4] OR RestoreAllToDefault OR di_LocalMode_setup.RestoreDefault) THEN (*Copy values into HMI variable and reset*)
	hmi_DiSetup[4]:=di_LocalMode_setup; (*Copy setup values from retain into hmi variable*)
	hmi_RestoreDefault_di[4]:=FALSE; (*Make sure that the restore variable is turned off after one restore command*)
	di_LocalMode_setup.RestoreDefault:=FALSE; (*Make sure that the restore variable is turned off after one restore command*)
END_IF
IF (hmi_DiWriteSetup[4]) THEN
	di_LocalMode_setup:=hmi_DiSetup[4]; (*Paste hmi changes back into setup variable*)
	hmi_DiWriteSetup[4]:=FALSE; (*Make sure that the write variable is turned off after one write command*)
END_IF
F_Trig[4](CLK:=hmi_DiPV[4].IsForced); (*Reset HMI forcing dialog when timer runs out*)
IF (F_Trig[4].Q) THEN hmi_DiSetup[4].Enable.Forcing:=FALSE;di_LocalMode_setup.Enable.Forcing:=FALSE; END_IF
(**************************************************)

(**************di_RemoteMode***********************)
IF (RestoreAllToDefault OR di_RemoteMode_setup.RestoreDefault  OR hmi_RestoreDefault_di[5]) THEN
	di_RemoteMode_setup.Name:='di_RemoteMode';
	di_RemoteMode_setup.CardNb:=PRG_HMI.setup_DioCard1_Number;
	di_RemoteMode_setup.ChannelMode:=1;
	di_RemoteMode_setup.ChannelNb:=18;
 	di_RemoteMode_setup.Delay.TOF:=T#0ms;
	di_RemoteMode_setup.Delay.TON:=T#0ms;
	di_RemoteMode_setup.Enable.Forcing:=0;
	di_RemoteMode_setup.Enable.TON:=0;
	di_RemoteMode_setup.Enable.TOF:=0;
	di_RemoteMode_setup.Levels.ForceValue:=0;
END_IF
IF (hmi_RestoreDefault_di[5] OR RestoreAllToDefault OR di_RemoteMode_setup.RestoreDefault) THEN (*Copy values into HMI variable and reset*)
	hmi_DiSetup[5]:=di_RemoteMode_setup; (*Copy setup values from retain into hmi variable*)
	hmi_RestoreDefault_di[5]:=FALSE; (*Make sure that the restore variable is turned off after one restore command*)
	di_RemoteMode_setup.RestoreDefault:=FALSE; (*Make sure that the restore variable is turned off after one restore command*)
END_IF
IF (hmi_DiWriteSetup[5]) THEN
	di_RemoteMode_setup:=hmi_DiSetup[5]; (*Paste hmi changes back into setup variable*)
	hmi_DiWriteSetup[5]:=FALSE; (*Make sure that the write variable is turned off after one write command*)
END_IF
F_Trig[5](CLK:=hmi_DiPV[5].IsForced); (*Reset HMI forcing dialog when timer runs out*)
IF (F_Trig[5].Q) THEN hmi_DiSetup[5].Enable.Forcing:=FALSE;di_RemoteMode_setup.Enable.Forcing:=FALSE; END_IF
(**************************************************)

(**************di_LocalStart***********************)
IF (RestoreAllToDefault OR di_LocalStart_setup.RestoreDefault  OR hmi_RestoreDefault_di[6]) THEN
	di_LocalStart_setup.Name:='di_LocalStart';
	di_LocalStart_setup.CardNb:=PRG_HMI.setup_DioCard1_Number;
	di_LocalStart_setup.ChannelMode:=1;
	di_LocalStart_setup.ChannelNb:=19;
 	di_LocalStart_setup.Delay.TOF:=T#0ms;
	di_LocalStart_setup.Delay.TON:=T#0ms;
	di_LocalStart_setup.Enable.Forcing:=0;
	di_LocalStart_setup.Enable.TON:=0;
	di_LocalStart_setup.Enable.TOF:=0;
	di_LocalStart_setup.Levels.ForceValue:=0;
END_IF
IF (hmi_RestoreDefault_di[6] OR RestoreAllToDefault OR di_LocalStart_setup.RestoreDefault) THEN (*Copy values into HMI variable and reset*)
	hmi_DiSetup[6]:=di_LocalStart_setup; (*Copy setup values from retain into hmi variable*)
	hmi_RestoreDefault_di[6]:=FALSE; (*Make sure that the restore variable is turned off after one restore command*)
	di_LocalStart_setup.RestoreDefault:=FALSE; (*Make sure that the restore variable is turned off after one restore command*)
END_IF
IF (hmi_DiWriteSetup[6]) THEN
	di_LocalStart_setup:=hmi_DiSetup[6]; (*Paste hmi changes back into setup variable*)
	hmi_DiWriteSetup[6]:=FALSE; (*Make sure that the write variable is turned off after one write command*)
END_IF
F_Trig[6](CLK:=hmi_DiPV[6].IsForced); (*Reset HMI forcing dialog when timer runs out*)
IF (F_Trig[6].Q) THEN hmi_DiSetup[6].Enable.Forcing:=FALSE;di_LocalStart_setup.Enable.Forcing:=FALSE; END_IF
(**************************************************)

(**************di_LocalStop***********************)
IF (RestoreAllToDefault OR di_LocalStop_setup.RestoreDefault  OR hmi_RestoreDefault_di[7]) THEN
	di_LocalStop_setup.Name:='di_LocalStop';
	di_LocalStop_setup.CardNb:=PRG_HMI.setup_DioCard1_Number;
	di_LocalStop_setup.ChannelMode:=1;
	di_LocalStop_setup.ChannelNb:=20;
 	di_LocalStop_setup.Delay.TOF:=T#0ms;
	di_LocalStop_setup.Delay.TON:=T#0ms;
	di_LocalStop_setup.Enable.Forcing:=0;
	di_LocalStop_setup.Enable.TON:=0;
	di_LocalStop_setup.Enable.TOF:=0;
	di_LocalStop_setup.Levels.ForceValue:=0;
END_IF
IF (hmi_RestoreDefault_di[7] OR RestoreAllToDefault OR di_LocalStop_setup.RestoreDefault) THEN (*Copy values into HMI variable and reset*)
	hmi_DiSetup[7]:=di_LocalStop_setup; (*Copy setup values from retain into hmi variable*)
	hmi_RestoreDefault_di[7]:=FALSE; (*Make sure that the restore variable is turned off after one restore command*)
	di_LocalStop_setup.RestoreDefault:=FALSE; (*Make sure that the restore variable is turned off after one restore command*)
END_IF
IF (hmi_DiWriteSetup[7]) THEN
	di_LocalStop_setup:=hmi_DiSetup[7]; (*Paste hmi changes back into setup variable*)
	hmi_DiWriteSetup[7]:=FALSE; (*Make sure that the write variable is turned off after one write command*)
END_IF
F_Trig[7](CLK:=hmi_DiPV[7].IsForced); (*Reset HMI forcing dialog when timer runs out*)
IF (F_Trig[7].Q) THEN hmi_DiSetup[7].Enable.Forcing:=FALSE;di_LocalStop_setup.Enable.Forcing:=FALSE; END_IF
(**************************************************)

(**************di_LocalReset***********************)
IF (RestoreAllToDefault OR di_LocalReset_setup.RestoreDefault  OR hmi_RestoreDefault_di[8]) THEN
	di_LocalReset_setup.Name:='di_LocalReset';
	di_LocalReset_setup.CardNb:=PRG_HMI.setup_DioCard1_Number;
	di_LocalReset_setup.ChannelMode:=1;
	di_LocalReset_setup.ChannelNb:=21;
 	di_LocalReset_setup.Delay.TOF:=T#0ms;
	di_LocalReset_setup.Delay.TON:=T#0ms;
	di_LocalReset_setup.Enable.Forcing:=0;
	di_LocalReset_setup.Enable.TON:=0;
	di_LocalReset_setup.Enable.TOF:=0;
	di_LocalReset_setup.Levels.ForceValue:=0;
END_IF
IF (hmi_RestoreDefault_di[8] OR RestoreAllToDefault OR di_LocalReset_setup.RestoreDefault) THEN (*Copy values into HMI variable and reset*)
	hmi_DiSetup[8]:=di_LocalReset_setup; (*Copy setup values from retain into hmi variable*)
	hmi_RestoreDefault_di[8]:=FALSE; (*Make sure that the restore variable is turned off after one restore command*)
	di_LocalReset_setup.RestoreDefault:=FALSE; (*Make sure that the restore variable is turned off after one restore command*)
END_IF
IF (hmi_DiWriteSetup[8]) THEN
	di_LocalReset_setup:=hmi_DiSetup[8]; (*Paste hmi changes back into setup variable*)
	hmi_DiWriteSetup[8]:=FALSE; (*Make sure that the write variable is turned off after one write command*)
END_IF
F_Trig[8](CLK:=hmi_DiPV[8].IsForced); (*Reset HMI forcing dialog when timer runs out*)
IF (F_Trig[8].Q) THEN hmi_DiSetup[8].Enable.Forcing:=FALSE;di_LocalReset_setup.Enable.Forcing:=FALSE; END_IF
(**************************************************)

(**************di_LocalEmergencyStop***********************)
IF (RestoreAllToDefault OR di_LocalEmergencyStop_setup.RestoreDefault  OR hmi_RestoreDefault_di[9]) THEN
	di_LocalEmergencyStop_setup.Name:='di_LocalEmergencyStop';
	di_LocalEmergencyStop_setup.CardNb:=PRG_HMI.setup_DioCard1_Number;
	di_LocalEmergencyStop_setup.ChannelMode:=1;
	di_LocalEmergencyStop_setup.ChannelNb:=22;
 	di_LocalEmergencyStop_setup.Delay.TOF:=T#0ms;
	di_LocalEmergencyStop_setup.Delay.TON:=T#0ms;
	di_LocalEmergencyStop_setup.Enable.Forcing:=0;
	di_LocalEmergencyStop_setup.Enable.TON:=0;
	di_LocalEmergencyStop_setup.Enable.TOF:=0;
	di_LocalEmergencyStop_setup.Levels.ForceValue:=0;
END_IF
IF (hmi_RestoreDefault_di[9] OR RestoreAllToDefault OR di_LocalEmergencyStop_setup.RestoreDefault) THEN (*Copy values into HMI variable and reset*)
	hmi_DiSetup[9]:=di_LocalEmergencyStop_setup; (*Copy setup values from retain into hmi variable*)
	hmi_RestoreDefault_di[9]:=FALSE; (*Make sure that the restore variable is turned off after one restore command*)
	di_LocalEmergencyStop_setup.RestoreDefault:=FALSE; (*Make sure that the restore variable is turned off after one restore command*)
END_IF
IF (hmi_DiWriteSetup[9]) THEN
	di_LocalEmergencyStop_setup:=hmi_DiSetup[9]; (*Paste hmi changes back into setup variable*)
	hmi_DiWriteSetup[9]:=FALSE; (*Make sure that the write variable is turned off after one write command*)
END_IF
F_Trig[9](CLK:=hmi_DiPV[9].IsForced); (*Reset HMI forcing dialog when timer runs out*)
IF (F_Trig[9].Q) THEN hmi_DiSetup[9].Enable.Forcing:=FALSE;di_LocalEmergencyStop_setup.Enable.Forcing:=FALSE; END_IF
(**************************************************)

(**************di_FusesOK***********************)
IF (RestoreAllToDefault OR di_FusesOK_setup.RestoreDefault  OR hmi_RestoreDefault_di[10]) THEN
	di_FusesOK_setup.Name:='di_FusesOK';
	di_FusesOK_setup.CardNb:=PRG_HMI.setup_DioCard1_Number;
	di_FusesOK_setup.ChannelMode:=1;
	di_FusesOK_setup.ChannelNb:=23;
 	di_FusesOK_setup.Delay.TOF:=T#0ms;
	di_FusesOK_setup.Delay.TON:=T#0ms;
	di_FusesOK_setup.Enable.Forcing:=0;
	di_FusesOK_setup.Enable.TON:=0;
	di_FusesOK_setup.Enable.TOF:=0;
	di_FusesOK_setup.Levels.ForceValue:=0;
END_IF
IF (hmi_RestoreDefault_di[10] OR RestoreAllToDefault OR di_FusesOK_setup.RestoreDefault) THEN (*Copy values into HMI variable and reset*)
	hmi_DiSetup[10]:=di_FusesOK_setup; (*Copy setup values from retain into hmi variable*)
	hmi_RestoreDefault_di[10]:=FALSE; (*Make sure that the restore variable is turned off after one restore command*)
	di_FusesOK_setup.RestoreDefault:=FALSE; (*Make sure that the restore variable is turned off after one restore command*)
END_IF
IF (hmi_DiWriteSetup[10]) THEN
	di_FusesOK_setup:=hmi_DiSetup[10]; (*Paste hmi changes back into setup variable*)
	hmi_DiWriteSetup[10]:=FALSE; (*Make sure that the write variable is turned off after one write command*)
END_IF
F_Trig[10](CLK:=hmi_DiPV[10].IsForced); (*Reset HMI forcing dialog when timer runs out*)
IF (F_Trig[10].Q) THEN hmi_DiSetup[10].Enable.Forcing:=FALSE;di_FusesOK_setup.Enable.Forcing:=FALSE; END_IF
(**************************************************)

(**************di_DcBreakerOpen***********************)
IF (RestoreAllToDefault OR di_DcBreakerOpen_setup.RestoreDefault  OR hmi_RestoreDefault_di[11]) THEN
	di_DcBreakerOpen_setup.Name:='di_DcBreakerOpen';
	di_DcBreakerOpen_setup.CardNb:=PRG_HMI.setup_DioCard1_Number;
	di_DcBreakerOpen_setup.ChannelMode:=1;
	di_DcBreakerOpen_setup.ChannelNb:=24;
 	di_DcBreakerOpen_setup.Delay.TOF:=T#0ms;
	di_DcBreakerOpen_setup.Delay.TON:=T#0ms;
	di_DcBreakerOpen_setup.Enable.Forcing:=0;
	di_DcBreakerOpen_setup.Enable.TON:=0;
	di_DcBreakerOpen_setup.Enable.TOF:=0;
	di_DcBreakerOpen_setup.Levels.ForceValue:=0;
END_IF
IF (hmi_RestoreDefault_di[11] OR RestoreAllToDefault OR di_DcBreakerOpen_setup.RestoreDefault) THEN (*Copy values into HMI variable and reset*)
	hmi_DiSetup[11]:=di_DcBreakerOpen_setup; (*Copy setup values from retain into hmi variable*)
	hmi_RestoreDefault_di[11]:=FALSE; (*Make sure that the restore variable is turned off after one restore command*)
	di_DcBreakerOpen_setup.RestoreDefault:=FALSE; (*Make sure that the restore variable is turned off after one restore command*)
END_IF
IF (hmi_DiWriteSetup[11]) THEN
	di_DcBreakerOpen_setup:=hmi_DiSetup[11]; (*Paste hmi changes back into setup variable*)
	hmi_DiWriteSetup[11]:=FALSE; (*Make sure that the write variable is turned off after one write command*)
END_IF
F_Trig[11](CLK:=hmi_DiPV[11].IsForced); (*Reset HMI forcing dialog when timer runs out*)
IF (F_Trig[11].Q) THEN hmi_DiSetup[11].Enable.Forcing:=FALSE;di_DcBreakerOpen_setup.Enable.Forcing:=FALSE; END_IF
(**************************************************)

(**************di_DcBreakerClosed***********************)
IF (RestoreAllToDefault OR di_DcBreakerClosed_setup.RestoreDefault  OR hmi_RestoreDefault_di[12]) THEN
	di_DcBreakerClosed_setup.Name:='di_DcBreakerClosed';
	di_DcBreakerClosed_setup.CardNb:=PRG_HMI.setup_DioCard1_Number;
	di_DcBreakerClosed_setup.ChannelMode:=1;
	di_DcBreakerClosed_setup.ChannelNb:=25;
 	di_DcBreakerClosed_setup.Delay.TOF:=T#0ms;
	di_DcBreakerClosed_setup.Delay.TON:=T#0ms;
	di_DcBreakerClosed_setup.Enable.Forcing:=0;
	di_DcBreakerClosed_setup.Enable.TON:=0;
	di_DcBreakerClosed_setup.Enable.TOF:=0;
	di_DcBreakerClosed_setup.Levels.ForceValue:=0;
END_IF
IF (hmi_RestoreDefault_di[12] OR RestoreAllToDefault OR di_DcBreakerClosed_setup.RestoreDefault) THEN (*Copy values into HMI variable and reset*)
	hmi_DiSetup[12]:=di_DcBreakerClosed_setup; (*Copy setup values from retain into hmi variable*)
	hmi_RestoreDefault_di[12]:=FALSE; (*Make sure that the restore variable is turned off after one restore command*)
	di_DcBreakerClosed_setup.RestoreDefault:=FALSE; (*Make sure that the restore variable is turned off after one restore command*)
END_IF
IF (hmi_DiWriteSetup[12]) THEN
	di_DcBreakerClosed_setup:=hmi_DiSetup[12]; (*Paste hmi changes back into setup variable*)
	hmi_DiWriteSetup[12]:=FALSE; (*Make sure that the write variable is turned off after one write command*)
END_IF
F_Trig[12](CLK:=hmi_DiPV[12].IsForced); (*Reset HMI forcing dialog when timer runs out*)
IF (F_Trig[12].Q) THEN hmi_DiSetup[12].Enable.Forcing:=FALSE;di_DcBreakerClosed_setup.Enable.Forcing:=FALSE; END_IF
(**************************************************)

(**************di_EthernetSwitchAlarm***********************)
IF (RestoreAllToDefault OR di_EthernetSwitchAlarm_setup.RestoreDefault  OR hmi_RestoreDefault_di[13]) THEN
	di_EthernetSwitchAlarm_setup.Name:='di_EthernetSwitchAlarm';
	di_EthernetSwitchAlarm_setup.CardNb:=PRG_HMI.setup_DioCard1_Number;
	di_EthernetSwitchAlarm_setup.ChannelMode:=1;
	di_EthernetSwitchAlarm_setup.ChannelNb:=26;
 	di_EthernetSwitchAlarm_setup.Delay.TOF:=T#0ms;
	di_EthernetSwitchAlarm_setup.Delay.TON:=T#0ms;
	di_EthernetSwitchAlarm_setup.Enable.Forcing:=0;
	di_EthernetSwitchAlarm_setup.Enable.TON:=0;
	di_EthernetSwitchAlarm_setup.Enable.TOF:=0;
	di_EthernetSwitchAlarm_setup.Levels.ForceValue:=0;
END_IF
IF (hmi_RestoreDefault_di[13] OR RestoreAllToDefault OR di_EthernetSwitchAlarm_setup.RestoreDefault) THEN (*Copy values into HMI variable and reset*)
	hmi_DiSetup[13]:=di_EthernetSwitchAlarm_setup; (*Copy setup values from retain into hmi variable*)
	hmi_RestoreDefault_di[13]:=FALSE; (*Make sure that the restore variable is turned off after one restore command*)
	di_EthernetSwitchAlarm_setup.RestoreDefault:=FALSE; (*Make sure that the restore variable is turned off after one restore command*)
END_IF
IF (hmi_DiWriteSetup[13]) THEN
	di_EthernetSwitchAlarm_setup:=hmi_DiSetup[13]; (*Paste hmi changes back into setup variable*)
	hmi_DiWriteSetup[13]:=FALSE; (*Make sure that the write variable is turned off after one write command*)
END_IF
F_Trig[13](CLK:=hmi_DiPV[13].IsForced); (*Reset HMI forcing dialog when timer runs out*)
IF (F_Trig[13].Q) THEN hmi_DiSetup[13].Enable.Forcing:=FALSE;di_EthernetSwitchAlarm_setup.Enable.Forcing:=FALSE; END_IF
(**************************************************)

(**************di_EmergencyStopLoopFault***********************)
IF (RestoreAllToDefault OR di_EmergencyStopLoopFault_setup.RestoreDefault  OR hmi_RestoreDefault_di[14]) THEN
	di_EmergencyStopLoopFault_setup.Name:='di_EmergencyStopLoopFault';
	di_EmergencyStopLoopFault_setup.CardNb:=PRG_HMI.setup_DioCard1_Number;
	di_EmergencyStopLoopFault_setup.ChannelMode:=1;
	di_EmergencyStopLoopFault_setup.ChannelNb:=27;
 	di_EmergencyStopLoopFault_setup.Delay.TOF:=T#0ms;
	di_EmergencyStopLoopFault_setup.Delay.TON:=T#0ms;
	di_EmergencyStopLoopFault_setup.Enable.Forcing:=0;
	di_EmergencyStopLoopFault_setup.Enable.TON:=0;
	di_EmergencyStopLoopFault_setup.Enable.TOF:=0;
	di_EmergencyStopLoopFault_setup.Levels.ForceValue:=0;
END_IF
IF (hmi_RestoreDefault_di[14] OR RestoreAllToDefault OR di_EmergencyStopLoopFault_setup.RestoreDefault) THEN (*Copy values into HMI variable and reset*)
	hmi_DiSetup[14]:=di_EmergencyStopLoopFault_setup; (*Copy setup values from retain into hmi variable*)
	hmi_RestoreDefault_di[14]:=FALSE; (*Make sure that the restore variable is turned off after one restore command*)
	di_EmergencyStopLoopFault_setup.RestoreDefault:=FALSE; (*Make sure that the restore variable is turned off after one restore command*)
END_IF
IF (hmi_DiWriteSetup[14]) THEN
	di_EmergencyStopLoopFault_setup:=hmi_DiSetup[14]; (*Paste hmi changes back into setup variable*)
	hmi_DiWriteSetup[14]:=FALSE; (*Make sure that the write variable is turned off after one write command*)
END_IF
F_Trig[14](CLK:=hmi_DiPV[14].IsForced); (*Reset HMI forcing dialog when timer runs out*)
IF (F_Trig[14].Q) THEN hmi_DiSetup[14].Enable.Forcing:=FALSE;di_EmergencyStopLoopFault_setup.Enable.Forcing:=FALSE; END_IF
(**************************************************)

(**************di_BatteryAuxOK***********************)
IF (RestoreAllToDefault OR di_BatteryAuxOK_setup.RestoreDefault  OR hmi_RestoreDefault_di[15]) THEN
	di_BatteryAuxOK_setup.Name:='di_BatteryAuxOK';
	di_BatteryAuxOK_setup.CardNb:=PRG_HMI.setup_DioCard1_Number;
	di_BatteryAuxOK_setup.ChannelMode:=1;
	di_BatteryAuxOK_setup.ChannelNb:=28;
 	di_BatteryAuxOK_setup.Delay.TOF:=T#0ms;
	di_BatteryAuxOK_setup.Delay.TON:=T#0ms;
	di_BatteryAuxOK_setup.Enable.Forcing:=0;
	di_BatteryAuxOK_setup.Enable.TON:=0;
	di_BatteryAuxOK_setup.Enable.TOF:=0;
	di_BatteryAuxOK_setup.Levels.ForceValue:=0;
END_IF
IF (hmi_RestoreDefault_di[15] OR RestoreAllToDefault OR di_BatteryAuxOK_setup.RestoreDefault) THEN (*Copy values into HMI variable and reset*)
	hmi_DiSetup[15]:=di_BatteryAuxOK_setup; (*Copy setup values from retain into hmi variable*)
	hmi_RestoreDefault_di[15]:=FALSE; (*Make sure that the restore variable is turned off after one restore command*)
	di_BatteryAuxOK_setup.RestoreDefault:=FALSE; (*Make sure that the restore variable is turned off after one restore command*)
END_IF
IF (hmi_DiWriteSetup[15]) THEN
	di_BatteryAuxOK_setup:=hmi_DiSetup[15]; (*Paste hmi changes back into setup variable*)
	hmi_DiWriteSetup[15]:=FALSE; (*Make sure that the write variable is turned off after one write command*)
END_IF
F_Trig[15](CLK:=hmi_DiPV[15].IsForced); (*Reset HMI forcing dialog when timer runs out*)
IF (F_Trig[15].Q) THEN hmi_DiSetup[15].Enable.Forcing:=FALSE;di_BatteryAuxOK_setup.Enable.Forcing:=FALSE; END_IF
(**************************************************)

(**************di_BatteryAuxNotOK***********************)
IF (RestoreAllToDefault OR di_BatteryAuxNotOK_setup.RestoreDefault  OR hmi_RestoreDefault_di[16]) THEN
	di_BatteryAuxNotOK_setup.Name:='di_BatteryAuxNotOK';
	di_BatteryAuxNotOK_setup.CardNb:=PRG_HMI.setup_DioCard1_Number;
	di_BatteryAuxNotOK_setup.ChannelMode:=1;
	di_BatteryAuxNotOK_setup.ChannelNb:=29;
 	di_BatteryAuxNotOK_setup.Delay.TOF:=T#0ms;
	di_BatteryAuxNotOK_setup.Delay.TON:=T#0ms;
	di_BatteryAuxNotOK_setup.Enable.Forcing:=0;
	di_BatteryAuxNotOK_setup.Enable.TON:=0;
	di_BatteryAuxNotOK_setup.Enable.TOF:=0;
	di_BatteryAuxNotOK_setup.Levels.ForceValue:=0;
END_IF
IF (hmi_RestoreDefault_di[16] OR RestoreAllToDefault OR di_BatteryAuxNotOK_setup.RestoreDefault) THEN (*Copy values into HMI variable and reset*)
	hmi_DiSetup[16]:=di_BatteryAuxNotOK_setup; (*Copy setup values from retain into hmi variable*)
	hmi_RestoreDefault_di[16]:=FALSE; (*Make sure that the restore variable is turned off after one restore command*)
	di_BatteryAuxNotOK_setup.RestoreDefault:=FALSE; (*Make sure that the restore variable is turned off after one restore command*)
END_IF
IF (hmi_DiWriteSetup[16]) THEN
	di_BatteryAuxNotOK_setup:=hmi_DiSetup[16]; (*Paste hmi changes back into setup variable*)
	hmi_DiWriteSetup[16]:=FALSE; (*Make sure that the write variable is turned off after one write command*)
END_IF
F_Trig[16](CLK:=hmi_DiPV[16].IsForced); (*Reset HMI forcing dialog when timer runs out*)
IF (F_Trig[16].Q) THEN hmi_DiSetup[16].Enable.Forcing:=FALSE;di_BatteryAuxNotOK_setup.Enable.Forcing:=FALSE; END_IF
(**************************************************)

(**************di_WaterLeakageDetected***********************)
IF (RestoreAllToDefault OR di_WaterLeakageDetected_setup.RestoreDefault  OR hmi_RestoreDefault_di[17]) THEN
	di_WaterLeakageDetected_setup.Name:='di_WaterLeakageDetected';
	di_WaterLeakageDetected_setup.CardNb:=PRG_HMI.setup_DioCard1_Number;
	di_WaterLeakageDetected_setup.ChannelMode:=1;
	di_WaterLeakageDetected_setup.ChannelNb:=30;
 	di_WaterLeakageDetected_setup.Delay.TOF:=T#0ms;
	di_WaterLeakageDetected_setup.Delay.TON:=T#0ms;
	di_WaterLeakageDetected_setup.Enable.Forcing:=0;
	di_WaterLeakageDetected_setup.Enable.TON:=0;
	di_WaterLeakageDetected_setup.Enable.TOF:=0;
	di_WaterLeakageDetected_setup.Levels.ForceValue:=0;
END_IF
IF (hmi_RestoreDefault_di[17] OR RestoreAllToDefault OR di_WaterLeakageDetected_setup.RestoreDefault) THEN (*Copy values into HMI variable and reset*)
	hmi_DiSetup[17]:=di_WaterLeakageDetected_setup; (*Copy setup values from retain into hmi variable*)
	hmi_RestoreDefault_di[17]:=FALSE; (*Make sure that the restore variable is turned off after one restore command*)
	di_WaterLeakageDetected_setup.RestoreDefault:=FALSE; (*Make sure that the restore variable is turned off after one restore command*)
END_IF
IF (hmi_DiWriteSetup[17]) THEN
	di_WaterLeakageDetected_setup:=hmi_DiSetup[17]; (*Paste hmi changes back into setup variable*)
	hmi_DiWriteSetup[17]:=FALSE; (*Make sure that the write variable is turned off after one write command*)
END_IF
F_Trig[17](CLK:=hmi_DiPV[17].IsForced); (*Reset HMI forcing dialog when timer runs out*)
IF (F_Trig[17].Q) THEN hmi_DiSetup[17].Enable.Forcing:=FALSE;di_WaterLeakageDetected_setup.Enable.Forcing:=FALSE; END_IF
(**************************************************)

(**************di_RemoteEmergencyStop***********************)
IF (RestoreAllToDefault OR di_RemoteEmergencyStop_setup.RestoreDefault  OR hmi_RestoreDefault_di[18]) THEN
	di_RemoteEmergencyStop_setup.Name:='di_RemoteEmergencyStop';
	di_RemoteEmergencyStop_setup.CardNb:=PRG_HMI.setup_DioCard1_Number;
	di_RemoteEmergencyStop_setup.ChannelMode:=1;
	di_RemoteEmergencyStop_setup.ChannelNb:=31;
 	di_RemoteEmergencyStop_setup.Delay.TOF:=T#0ms;
	di_RemoteEmergencyStop_setup.Delay.TON:=T#0ms;
	di_RemoteEmergencyStop_setup.Enable.Forcing:=0;
	di_RemoteEmergencyStop_setup.Enable.TON:=0;
	di_RemoteEmergencyStop_setup.Enable.TOF:=0;
	di_RemoteEmergencyStop_setup.Levels.ForceValue:=0;
END_IF
IF (hmi_RestoreDefault_di[18] OR RestoreAllToDefault OR di_RemoteEmergencyStop_setup.RestoreDefault) THEN (*Copy values into HMI variable and reset*)
	hmi_DiSetup[18]:=di_RemoteEmergencyStop_setup; (*Copy setup values from retain into hmi variable*)
	hmi_RestoreDefault_di[18]:=FALSE; (*Make sure that the restore variable is turned off after one restore command*)
	di_RemoteEmergencyStop_setup.RestoreDefault:=FALSE; (*Make sure that the restore variable is turned off after one restore command*)
END_IF
IF (hmi_DiWriteSetup[18]) THEN
	di_RemoteEmergencyStop_setup:=hmi_DiSetup[18]; (*Paste hmi changes back into setup variable*)
	hmi_DiWriteSetup[18]:=FALSE; (*Make sure that the write variable is turned off after one write command*)
END_IF
F_Trig[18](CLK:=hmi_DiPV[18].IsForced); (*Reset HMI forcing dialog when timer runs out*)
IF (F_Trig[18].Q) THEN hmi_DiSetup[18].Enable.Forcing:=FALSE;di_RemoteEmergencyStop_setup.Enable.Forcing:=FALSE; END_IF
(**************************************************)

(**************di_SpareChannel32***********************)
IF (RestoreAllToDefault OR di_SpareChannel32_setup.RestoreDefault  OR hmi_RestoreDefault_di[19]) THEN
	di_SpareChannel32_setup.Name:='di_SpareChannel32';
	di_SpareChannel32_setup.CardNb:=PRG_HMI.setup_DioCard1_Number;
	di_SpareChannel32_setup.ChannelMode:=1;
	di_SpareChannel32_setup.ChannelNb:=32;
 	di_SpareChannel32_setup.Delay.TOF:=T#0ms;
	di_SpareChannel32_setup.Delay.TON:=T#0ms;
	di_SpareChannel32_setup.Enable.Forcing:=0;
	di_SpareChannel32_setup.Enable.TON:=0;
	di_SpareChannel32_setup.Enable.TOF:=0;
	di_SpareChannel32_setup.Levels.ForceValue:=0;
END_IF
IF (hmi_RestoreDefault_di[19] OR RestoreAllToDefault OR di_SpareChannel32_setup.RestoreDefault) THEN (*Copy values into HMI variable and reset*)
	hmi_DiSetup[19]:=di_SpareChannel32_setup; (*Copy setup values from retain into hmi variable*)
	hmi_RestoreDefault_di[19]:=FALSE; (*Make sure that the restore variable is turned off after one restore command*)
	di_SpareChannel32_setup.RestoreDefault:=FALSE; (*Make sure that the restore variable is turned off after one restore command*)
END_IF
IF (hmi_DiWriteSetup[19]) THEN
	di_SpareChannel32_setup:=hmi_DiSetup[19]; (*Paste hmi changes back into setup variable*)
	hmi_DiWriteSetup[19]:=FALSE; (*Make sure that the write variable is turned off after one write command*)
END_IF
F_Trig[19](CLK:=hmi_DiPV[19].IsForced); (*Reset HMI forcing dialog when timer runs out*)
IF (F_Trig[19].Q) THEN hmi_DiSetup[19].Enable.Forcing:=FALSE;di_SpareChannel32_setup.Enable.Forcing:=FALSE; END_IF
(**************************************************)

END_ACTION

END_ACTIONS
